Universal Robots URScript: samho_main_Fillet_2023_10_18.script

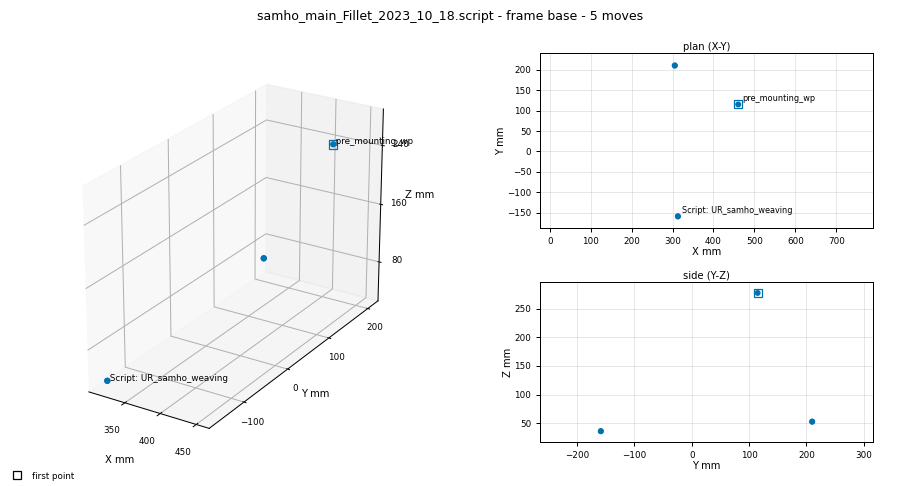
[picture p0: tool path of samho_main_Fillet_2023_10_18.script in frame base, 5 of 118 moves have a stored position in this frame; points joined in program order, loops and branches not executed]
def samho_main_Fillet_2023_10_18():
  set_standard_analog_input_domain(0, 1)
  set_standard_analog_input_domain(1, 1)
  set_tool_analog_input_domain(0, 1)
  set_tool_analog_input_domain(1, 1)
  set_analog_outputdomain(0, 1)
  set_analog_outputdomain(1, 1)
  set_input_actions_to_default()
  set_tool_digital_input_action(1, "freedrive")
  set_runstate_standard_digital_outputs([0])
  set_runstate_standard_digital_output_to_value(0, 1)
  set_runstate_standard_digital_output_to_value(7, 3)
  step_count_71f140af_8f37_405c_9852_4a67516a149e = 0.0
  thread Step_Counter_Thread_85a6b8af_9cee_45e5_b399_1c83c9369c53():
    while (True):
      step_count_71f140af_8f37_405c_9852_4a67516a149e = step_count_71f140af_8f37_405c_9852_4a67516a149e + 1.0
      sync()
    end
  end
  run Step_Counter_Thread_85a6b8af_9cee_45e5_b399_1c83c9369c53()
  modbus_add_signal("127.0.0.1", 255, 142, 2, "MODBUS_1", False)
  modbus_set_signal_update_frequency("MODBUS_1", 1)
  modbus_add_signal("127.0.0.1", 255, 152, 2, "MODBUS_2", False)
  modbus_set_signal_update_frequency("MODBUS_2", 10)
  modbus_add_signal("127.0.0.1", 255, 153, 2, "MODBUS_3", False)
  modbus_set_signal_update_frequency("MODBUS_3", 10)
  modbus_add_signal("127.0.0.1", 255, 240, 2, "MODBUS_4", False)
  modbus_set_signal_update_frequency("MODBUS_4", 10)
  set_safety_mode_transition_hardness(1)
  set_tool_voltage(24)
  set_tcp(p[-0.20862,-0.00524,0.38449,1.2551,0.019,-2.8747])
  set_payload(2.4, [-0.085, 0.00191, 0.125])
  set_gravity([0.0, 0.0, 9.82])
  global A_Touch_trig_l=[False, True, False, True, False, True, False, True, False, False, False]
  global Auto_cur_cell=0
  global last_wv_line=p[0, 0, 0, 0, 0, 0]
  global Auto_trig=True
  global A_Touch_p=[p[0, 0, 0, 0, 0, 0], p[0.49652, 0.34473, -0.02809, -1.74217, -0.74593, -1.74161], p[0, 0, 0, 0, 0, 0], p[0.50294, -0.36001, 0.02477, 1.70888, -0.78236, 1.70938], p[0, 0, 0, 0, 0, 0], p[0.49786, 0.33965, -0.0331, -1.74681, 1.75003, -0.74209], p[0, 0, 0, 0, 0, 0], p[0.50148, -0.2752, -0.03447, -1.75566, 1.75559, -0.7328], p[0, 0, 0, 0, 0, 0], p[0, 0, 0, 0, 0, 0], p[0, 0, 0, 0, 0, 0], p[0, 0, 0, 0, 0, 0], p[0, 0, 0, 0, 0, 0], p[0, 0, 0, 0, 0, 0], p[0, 0, 0, 0, 0, 0], p[0, 0, 0, 0, 0, 0]]
  global last_wv_wp1=p[0, 0, 0, 0, 0, 0]
  global last_pose=p[0, 0, 0, 0, 0, 0]
  global A_Distance_list=[0, 0, 0, 0, 0, 0, 0, 0, 0, 0, 0, 0, 0, 0, 0, 0]
  global Auto_total_cell=4
  global Reset_Trig=False
  global A_Prepos_l=[p[0, 0, 0, 0, 0, 0], p[0.46861, 0.32973, 0.0248, -2.17926, -0.88648, -1.41868], p[0, 0, 0, 0, 0, 0], p[0.46861, -0.33027, 0.0498, 1.84179, -1.10813, 1.58337], p[0, 0, 0, 0, 0, 0], p[0.47174, 0.31972, 0.02458, -2.36882, -1.02821, -1.3113], p[0, 0, 0, 0, 0, 0], p[0.46616, -0.25026, 0.02497, 2.26908, -1.08882, 1.27698], p[0, 0, 0, 0, 0, 0], p[0, 0, 0, 0, 0, 0], p[0, 0, 0, 0, 0, 0], p[0, 0, 0, 0, 0, 0], p[0, 0, 0, 0, 0, 0], p[0, 0, 0, 0, 0, 0], p[0, 0, 0, 0, 0, 0], p[0, 0, 0, 0, 0, 0]]
  global A_Speed_list=[0, 0, 0, 0, 0, 0, 0, 0, 0, 0, 0, 0, 0, 0, 0, 0]
  global Auto_W_num=[31, 32, 1, 3, 0, 0, 0, 0, 0, 0, 0, 0, 0, 0, 0]
  global last_z_bottom=-0.0502
  global last_tilt_deg=[0, 0, 0]
  global Base=p[0.0,0.0,0.0,0.0,0.0,0.0]
  global save_timer=0
  global timer_1=0
  def calculate_point_to_move_towards(feature, direction, position_distance):
    local posDir=[direction[0], direction[1], direction[2]]
    if (norm(posDir) < 1e-6):
      return get_target_waypoint()
    end
    local direction_vector_normalized=normalize(posDir)
    local displacement_pose=p[direction_vector_normalized[0] * position_distance,direction_vector_normalized[1] * position_distance,direction_vector_normalized[2] * position_distance,0,0,0]
    local wanted_displacement_in_base_frame=pose_sub(pose_trans(feature, displacement_pose), feature)
    return pose_add(get_target_waypoint(), wanted_displacement_in_base_frame)
  end
  global save_timer_is_counting=False
  global timer_1_is_counting=False
  thread Timer_Thread():
    while (True):
      if (save_timer_is_counting):
        save_timer = save_timer + get_steptime()
      end
      if (timer_1_is_counting):
        timer_1 = timer_1 + get_steptime()
      end
      sync()
    end
  end
  run Timer_Thread()
  def cell_info():
    $ 1461 "cell_info" "noBreak"
    $ 1462 "'cell_setting'"
    # 'cell_setting'
    $ 1463 "a7_f_distance≔get_center"
    global a7_f_distance=get_center
    $ 1464 "'dis + 125'"
    # 'dis + 125'
    $ 1465 "If simulation_mode"
    if (simulation_mode):
      $ 1466 "a6_f_height_l≔190"
      global a6_f_height_l=190
      $ 1467 "a6_f_height_r≔190"
      global a6_f_height_r=190
      $ 1468 "a6_f_width≔690"
      global a6_f_width=690
      $ 1469 "a6_callar_hor≔100"
      global a6_callar_hor=100
      $ 1470 "a6_callar_vert≔100"
      global a6_callar_vert=100
      $ 1471 "center_height≔50"
      global center_height=50
      $ 1472 "EXT_flag1≔integer_to_binary_list(2048)"
      global EXT_flag1= integer_to_binary_list (2048)
      $ 1473 "get_margin_z≔50"
      global get_margin_z=50
    else:
      $ 1474 "Else" "noBreak"
      $ 1475 "a6_f_height_l≔read_port_register(173)"
      global a6_f_height_l= read_port_register (173)
      $ 1476 "a6_f_height_r≔read_port_register(174)"
      global a6_f_height_r= read_port_register (174)
      $ 1477 "a6_f_width≔read_port_register(175)"
      global a6_f_width= read_port_register (175)
      $ 1478 "a6_callar_hor≔read_port_register(181)"
      global a6_callar_hor= read_port_register (181)
      $ 1479 "a6_callar_vert≔read_port_register(182)"
      global a6_callar_vert= read_port_register (182)
      $ 1480 "center_height≔read_port_register(237)"
      global center_height=read_port_register(237)
      $ 1481 "EXT_flag1≔integer_to_binary_list(read_port_register(179))"
      global EXT_flag1= integer_to_binary_list ( read_port_register (179))
      $ 1483 "get_margin_z≔read_port_register(238)"
      global get_margin_z=read_port_register(238)
      $ 1485 "If center_height>32765"
      if (center_height>32765):
        $ 1486 "center_height≔center_height-65535"
        global center_height=center_height-65535
      end
      $ 1487 "If get_margin_z>32765"
      if (get_margin_z>32765):
        $ 1488 "get_margin_z≔get_margin_z-65535"
        global get_margin_z=get_margin_z-65535
      end
    end
    $ 1489 "Initialization"
    $ 1490 "CELL_ROBOT_DIST≔a7_f_distance"
    global CELL_ROBOT_DIST=a7_f_distance
    $ 1491 "CELL_WIDTH≔a6_f_width"
    global CELL_WIDTH=a6_f_width
  end
  def robotand_cell_initalizat():
    $ 1492 "robotand_cell_initalizat" "noBreak"
    $ 1493 "If Auto_trig≟ True "
    if (Auto_trig ==   True  ):
      $ 1494 "Auto_trig≔ False "
      global Auto_trig=  False
      $ 1495 "init"
      $ 1496 "write_port_register(cell_3f_2f_151,0)"
      write_port_register(cell_3f_2f_151,0)
      $ 1497 "write_port_register(cell_info_152,0)"
      write_port_register(cell_info_152,0)
      $ 1498 "write_port_register(weld_req_153,0)"
      write_port_register(weld_req_153,0)
      $ 1499 "write_port_register(touch_cell_155,0)"
      write_port_register(touch_cell_155,0)
      $ 1500 "write_port_register(touch_num_156,0)"
      write_port_register(touch_num_156,0)
      $ 1501 "write_port_register(touch_done_157,0)"
      write_port_register(touch_done_157,0)
      $ 1502 "write_port_register(weld_done_137,0)"
      write_port_register(weld_done_137,0)
      $ 1503 "write_port_register(135,0)"
      write_port_register(135,0)
      $ 1504 "write_port_register(136,0)"
      write_port_register(136,0)
      $ 1505 "write_port_register(165,0)"
      write_port_register(165,0)
      $ 1506 "write_port_register(166,0)"
      write_port_register(166,0)
      $ 1507 "write_port_register(167,0)"
      write_port_register(167,0)
      $ 1508 "write_port_register(169,0)"
      write_port_register(169,0)
      $ 1509 "write_port_register(170,0)"
      write_port_register(170,0)
      $ 1510 "write_port_register(221,0)"
      write_port_register(221,0)
      $ 1511 "write_port_register(222,0)"
      write_port_register(222,0)
      $ 1512 "write_port_register(223,0)"
      write_port_register(223,0)
      $ 1513 "write_port_register(224,0)"
      write_port_register(224,0)
      $ 1514 "write_port_register(225,0)"
      write_port_register(225,0)
      $ 1515 "write_port_register(226,0)"
      write_port_register(226,0)
      $ 1516 "write_port_register(227,0)"
      write_port_register(227,0)
      $ 1517 "write_port_register(228,0)"
      write_port_register(228,0)
      $ 1518 "write_port_register(240,0)"
      write_port_register(240,0)
      $ 1519 "write_port_register(176,0)"
      write_port_register(176,0)
      $ 1520 "write_port_register(177,0)"
      write_port_register(177,0)
      $ 1521 "write_port_register(154,0)"
      write_port_register(154,0)
    end
    $ 1522 "sync()"
    sync()
  end
  def welding_parameter_init():
    $ 1523 "welding_parameter_init" "noBreak"
    $ 1524 "init"
    $ 1525 "If A_sel_v≟A_VL1 or A_sel_v≟A_VL2 or A_sel_v≟A_VR1 or A_sel_v≟A_VR2"
    if (A_sel_v == A_VL1  or  A_sel_v == A_VL2  or  A_sel_v == A_VR1  or  A_sel_v == A_VR2):
      $ 1526 "position_3f2f≔position_3F"
      global position_3f2f=position_3F
      $ 1527 "write_port_register(cell_3f_2f_151,A_sel_v)"
      write_port_register(cell_3f_2f_151,A_sel_v)
      $ 1528 "b8_wv_2f≔ False "
      global b8_wv_2f=  False
      $ 1529 "d_lean_degree≔0"
      global d_lean_degree=0
    else:
      $ 1530 "Else" "noBreak"
      $ 1531 "position_3f2f≔position_2F"
      global position_3f2f=position_2F
      $ 1532 "b8_wv_2f≔ True "
      global b8_wv_2f=  True
      $ 1533 "d_lean_degree≔30"
      global d_lean_degree=30
      $ 1534 "write_port_register(cell_3f_2f_151,A_HOR)"
      write_port_register(cell_3f_2f_151,A_HOR)
    end
    $ 1535 "If current_path≥2"
    if (current_path >= 2):
      $ 1536 "write_port_register(cell_info_152,current_path)"
      write_port_register(cell_info_152,current_path)
    else:
      $ 1537 "Else" "noBreak"
      $ 1538 "write_port_register(cell_info_152,1)"
      write_port_register(cell_info_152,1)
    end
    $ 1539 "write_port_register(return_done_240,0)"
    write_port_register(return_done_240,0)
    $ 1540 "Wait: 0.3"
    sleep(0.3)
    $ 1541 "write_port_register(weld_req_153,1)"
    write_port_register(weld_req_153,1)
    $ 1542 "Wait read_port_register(return_done_240)≟1"
    while (not( read_port_register (return_done_240) == 1)):
      sync()
    end
    $ 1543 "write_port_register(weld_req_153,0)"
    write_port_register(weld_req_153,0)
    $ 1544 "touch_m_check≔0"
    global touch_m_check=0
    $ 1545 "start_end_from_pendant"
    $ 1546 "d_start_current≔read_port_register(244)/10"
    global d_start_current= read_port_register (244)/10
    $ 1547 "d_start_voltage≔read_port_register(245)/10"
    global d_start_voltage= read_port_register (245)/10
    $ 1548 "d_start_time≔read_port_register(241)/10"
    global d_start_time= read_port_register (241)/10
    $ 1549 "d_end_current≔read_port_register(249)/10"
    global d_end_current= read_port_register (249)/10
    $ 1550 "d_end_voltage≔read_port_register(250)/10"
    global d_end_voltage= read_port_register (250)/10
    $ 1551 "d_end_time≔read_port_register(246)/10"
    global d_end_time= read_port_register (246)/10
    $ 1552 "d_end_current_2≔read_port_register(254)/10"
    global d_end_current_2= read_port_register (254)/10
    $ 1553 "d_end_voltage_2≔read_port_register(255)/10"
    global d_end_voltage_2= read_port_register (255)/10
    $ 1554 "d_end_time_2≔read_port_register(251)/10"
    global d_end_time_2= read_port_register (251)/10
    $ 1555 "a7_weld_crater≔[d_start_current,d_start_voltage,d_start_time,d_end_current,d_end_voltage,d_end_time,d_lean_degree]"
    global a7_weld_crater=[d_start_current,d_start_voltage,d_start_time,d_end_current,d_end_voltage,d_end_time,d_lean_degree]
    $ 1556 "a0_volt_ref≔read_port_register(231)/10"
    global a0_volt_ref= read_port_register (231)/10
    $ 1557 "a1_amp_ref≔read_port_register(232)/10"
    global a1_amp_ref= read_port_register (232)/10
    $ 1558 "a2_speed_cpm≔read_port_register(233)/10"
    global a2_speed_cpm= read_port_register (233)/10
    $ 1559 "a3_wv_amplitude≔read_port_register(234)/10"
    global a3_wv_amplitude= read_port_register (234)/10
    $ 1560 "a4_wv_frequency≔read_port_register(225)/10"
    global a4_wv_frequency= read_port_register (225)/10
    $ 1561 "b1_appro_param≔0"
    global b1_appro_param=0
    $ 1562 "b4_wv_delay2≔read_port_register(226)/10"
    global b4_wv_delay2= read_port_register (226)/10
    $ 1563 "b6_wv_delay4≔read_port_register(227)/10"
    global b6_wv_delay4= read_port_register (227)/10
    $ 1564 "b3_wv_delay1≔0"
    global b3_wv_delay1=0
    $ 1565 "b5_wv_delay3≔0"
    global b5_wv_delay3=0
    $ 1566 "b3_dealy_all≔[b3_wv_delay1,b4_wv_delay2,b5_wv_delay3,b6_wv_delay4]"
    global b3_dealy_all=[b3_wv_delay1,b4_wv_delay2,b5_wv_delay3,b6_wv_delay4]
    $ 1567 "get_width_182≔read_port_register(182)"
    global get_width_182= read_port_register (182)
    $ 1568 "b9_touch_sens≔20"
    global b9_touch_sens=20
    $ 1569 "task_angle≔register_read(228)/10"
    global task_angle=register_read(228)/10
    $ 1570 "Circle_Speed≔a2_speed_cpm"
    global Circle_Speed=a2_speed_cpm
    $ 1571 "CELL_BOTTOM≔a7_cell_bottom"
    global CELL_BOTTOM=a7_cell_bottom
    $ 1572 "a6_scallup_left≔read_port_register(176)"
    global a6_scallup_left= read_port_register (176)
    $ 1573 "a6_scallup_righ≔read_port_register(177)"
    global a6_scallup_righ= read_port_register (177)
    $ 1574 "a5_f_hole≔[a7_cell_bottom,a6_scallup_left,a6_scallup_righ]"
    global a5_f_hole=[a7_cell_bottom,a6_scallup_left,a6_scallup_righ]
    $ 1608 "폴더"
    $ 1609 "offset_2f_x≔7"
    global offset_2f_x=7
    $ 1610 "offset_3f_z≔-5"
    global offset_3f_z=-5
    $ 1611 "If A_sel_v≟A_VR1 or A_sel_v≟A_VR2"
    if (A_sel_v == A_VR1  or  A_sel_v == A_VR2):
      $ 1612 "'3F'"
      # '3F'
      $ 1613 "b2_left_par≔ False "
      global b2_left_par=  False
      $ 1614 "b8_wv_type≔1"
      global b8_wv_type=1
      $ 1615 "If A_sel_v≟A_VR2 and (b1_cell_info_R≟c or b1_cell_info_R≟d)"
      if (A_sel_v == A_VR2  and  (b1_cell_info_R == c  or  b1_cell_info_R == d)):
        $ 1616 "b7_tilt_degree≔[0,0,0]"
        global b7_tilt_degree=[0,0,0]
      else:
        $ 1617 "Else" "noBreak"
        $ 1618 "b7_tilt_degree≔[task_angle,-27,0]"
        global b7_tilt_degree=[task_angle,-27,0]
      end
      $ 1619 "c3_arc_enable≔1"
      global c3_arc_enable=1
    else:
      $ 1620 "ElseIf A_sel_v≟A_VL1 or A_sel_v≟A_VL2"
      if (A_sel_v == A_VL1  or  A_sel_v == A_VL2):
        $ 1621 "'3F'"
        # '3F'
        $ 1622 "b2_left_par≔ True "
        global b2_left_par=  True
        $ 1623 "b8_wv_type≔1"
        global b8_wv_type=1
        $ 1624 "If A_sel_v≟A_VL2 and (b1_cell_info_L≟c or b1_cell_info_L≟d)"
        if (A_sel_v == A_VL2  and  (b1_cell_info_L == c  or  b1_cell_info_L == d)):
          $ 1625 "b7_tilt_degree≔[0,0,0]"
          global b7_tilt_degree=[0,0,0]
        else:
          $ 1626 "Else" "noBreak"
          $ 1627 "b7_tilt_degree≔[task_angle,-27,0]"
          global b7_tilt_degree=[task_angle,-27,0]
        end
        $ 1628 "c3_arc_enable≔1"
        global c3_arc_enable=1
      else:
        $ 1629 "Else" "noBreak"
        $ 1630 "b2_left_par≔ True "
        global b2_left_par=  True
        $ 1631 "b8_wv_type≔2"
        global b8_wv_type=2
        $ 1632 "If A_sel_v≟A_HOR"
        if (A_sel_v == A_HOR):
          $ 1633 "b7_tilt_degree≔[30,-1*task_angle,0]"
          global b7_tilt_degree=[30,-1*task_angle,0]
        else:
          $ 1634 "Else" "noBreak"
          $ 1636 "b7_tilt_degree≔[30,-1*task_angle,0]"
          global b7_tilt_degree=[30,-1*task_angle,0]
        end
        $ 1638 "c3_arc_enable≔0"
        global c3_arc_enable=0
      end
    end
    $ 1639 "If A_sel_v≟A_VL2 or A_sel_v≟A_VR2"
    if (A_sel_v == A_VL2  or  A_sel_v == A_VR2):
      $ 1640 "a8_wv_distance≔read_port_register(182)-offset_3f_begin"
      global a8_wv_distance= read_port_register (182)-offset_3f_begin
    else:
      $ 1645 "Else" "noBreak"
      $ 1646 "If b2_left_par"
      if (b2_left_par):
        $ 1647 "Comment"
        # Comment
        $ 1648 "a8_wv_distance≔a6_f_height_l-a5_f_hole[1]-offset_3f_begin"
        global a8_wv_distance=a6_f_height_l-a5_f_hole[1]-offset_3f_begin
        $ 1649 "Comment"
        # Comment
      else:
        $ 1650 "Else" "noBreak"
        $ 1651 "a8_wv_distance≔a6_f_height_r-a5_f_hole[1]-offset_3f_begin"
        global a8_wv_distance=a6_f_height_r-a5_f_hole[1]-offset_3f_begin
      end
    end
    $ 1652 "Ext fun & Squash"
    $ 1653 "If (A_sel_v≟A_VL1 or A_sel_v≟A_VL2) and (b1_cell_info_L≟B or b1_cell_info_L≟D)"
    if ((A_sel_v == A_VL1  or  A_sel_v == A_VL2)  and  (b1_cell_info_L == B  or  b1_cell_info_L == D)):
      $ 1654 "Scallup_check≔ True "
      global Scallup_check=  True
    else:
      $ 1655 "ElseIf (A_sel_v≟A_VR1 or A_sel_v≟A_VR2) and (b1_cell_info_R≟B or b1_cell_info_R≟D)"
      if ((A_sel_v == A_VR1  or  A_sel_v == A_VR2)  and  (b1_cell_info_R == B  or  b1_cell_info_R == D)):
        $ 1656 "Scallup_check≔ True "
        global Scallup_check=  True
      else:
        $ 1657 "Else" "noBreak"
        $ 1658 "Scallup_check≔ False "
        global Scallup_check=  False
      end
    end
    $ 1659 "If (EXT_flag1[7]≟ True ) and (A_sel_v≠A_HOR) and (A_sel_v≠A_VL2) and (A_sel_v≠A_VR2) and (Scallup_check≟ False )"
    if ((EXT_flag1[7] ==   True  )  and  (A_sel_v != A_HOR)  and  (A_sel_v != A_VL2)  and  (A_sel_v != A_VR2)  and  (Scallup_check ==   False  )):
      $ 1660 "squash"
      $ 1661 "squash_enable≔1"
      global squash_enable=1
      $ 1662 "squash_voltage≔24.5"
      global squash_voltage=24.5
      $ 1663 "squash_current≔190"
      global squash_current=190
      $ 1664 "squash_amp≔7"
      global squash_amp=7
      $ 1665 "squash_speed≔10"
      global squash_speed=10
      $ 1666 "squash_cycle≔8"
      global squash_cycle=8
    else:
      $ 1667 "Else" "noBreak"
      $ 1668 "squash"
      $ 1669 "squash_enable≔0"
      global squash_enable=0
      $ 1670 "squash_voltage≔0"
      global squash_voltage=0
      $ 1671 "squash_current≔0"
      global squash_current=0
      $ 1672 "squash_amp≔0"
      global squash_amp=0
      $ 1673 "squash_speed≔0"
      global squash_speed=0
      $ 1674 "squash_cycle≔0"
      global squash_cycle=0
    end
    $ 1675 "If EXT_flag1[8]≟ True  and EXT_flag1[9]≟ False "
    if (EXT_flag1[8] ==   True    and  EXT_flag1[9] ==   False  ):
      $ 1676 "sludge≔1"
      global sludge=1
    else:
      $ 1677 "ElseIf EXT_flag1[8]≟ False  and EXT_flag1[9]≟ True "
      if (EXT_flag1[8] ==   False    and  EXT_flag1[9] ==   True  ):
        $ 1678 "sludge≔2"
        global sludge=2
      else:
        $ 1679 "Else" "noBreak"
        $ 1680 "sludge≔0"
        global sludge=0
      end
    end
    $ 1681 "waste_cycle≔2"
    global waste_cycle=2
    $ 1682 "c0_offset_x≔read_port_register(229)/10"
    global c0_offset_x= read_port_register (229)/10
    $ 1683 "c0_offset_z≔read_port_register(230)/10"
    global c0_offset_z= read_port_register (230)/10
    $ 1684 "squash_l≔[a0_volt_ref,a1_amp_ref,squash_enable,squash_voltage,squash_current,squash_amp,squash_speed,squash_cycle,waste_cycle,c0_offset_x,c0_offset_z]"
    global squash_l=[a0_volt_ref,a1_amp_ref,squash_enable,squash_voltage,squash_current,squash_amp,squash_speed,squash_cycle,waste_cycle,c0_offset_x,c0_offset_z]
    $ 1685 "WV_gap"
    $ 1686 "c5_wv_gap_y≔read_port_register(236)/10"
    global c5_wv_gap_y= read_port_register (236)/10
    $ 1687 "c6_wv_gap_cpm≔read_port_register(235)/10"
    global c6_wv_gap_cpm= read_port_register (235)/10
    $ 1688 "c9_wv_gap_freq≔a4_wv_frequency"
    global c9_wv_gap_freq=a4_wv_frequency
    $ 1689 "If c6_wv_gap_cpm≟a2_speed_cpm and a3_wv_amplitude≟c5_wv_gap_y"
    if (c6_wv_gap_cpm == a2_speed_cpm  and  a3_wv_amplitude == c5_wv_gap_y):
      $ 1690 "c4_gap_enable≔0"
      global c4_gap_enable=0
    else:
      $ 1691 "Else" "noBreak"
      $ 1692 "c4_gap_enable≔1"
      global c4_gap_enable=1
    end
    $ 1693 "c7_wv_gap≔[c4_gap_enable,c5_wv_gap_y,c6_wv_gap_cpm,c9_wv_gap_freq]"
    global c7_wv_gap=[c4_gap_enable,c5_wv_gap_y,c6_wv_gap_cpm,c9_wv_gap_freq]
    $ 1694 "arc_sen"
    $ 1695 "c3_X_p_gain≔read_port_register(186)/10"
    global c3_X_p_gain= read_port_register (186)/10
    $ 1696 "c3_X_i_gain≔read_port_register(187)/10"
    global c3_X_i_gain= read_port_register (187)/10
    $ 1697 "c3_Z_p_gain≔read_port_register(184)/10"
    global c3_Z_p_gain= read_port_register (184)/10
    $ 1698 "c3_Z_i_gain≔read_port_register(185)/10"
    global c3_Z_i_gain= read_port_register (185)/10
    $ 1699 "c3_wv_arc_fix≔0"
    global c3_wv_arc_fix=0
    $ 1700 "c3_wv_arc≔[c3_arc_enable,c3_X_p_gain,c3_X_i_gain,c3_Z_p_gain,c3_Z_i_gain,c3_wv_arc_fix]"
    global c3_wv_arc=[c3_arc_enable,c3_X_p_gain,c3_X_i_gain,c3_Z_p_gain,c3_Z_i_gain,c3_wv_arc_fix]
    $ 1701 "volt and current"
    $ 1702 "set_current_voltage(a1_amp_ref,a0_volt_ref)"
    set_current_voltage(a1_amp_ref,a0_volt_ref)
    $ 1703 "write_port_register(154,1)"
    write_port_register(154,1)
    $ 1704 "Wait read_port_register(return_done_240)≟0"
    while (not( read_port_register (return_done_240) == 0)):
      sync()
    end
    $ 1705 "write_port_register(154,0)"
    write_port_register(154,0)
  end
  def welding_parameter_sim():
    $ 1706 "welding_parameter_sim" "noBreak"
    $ 1707 "init"
    $ 1708 "If A_sel_v≟A_VL1 or A_sel_v≟A_VL2 or A_sel_v≟A_VR1 or A_sel_v≟A_VR2"
    if (A_sel_v == A_VL1  or  A_sel_v == A_VL2  or  A_sel_v == A_VR1  or  A_sel_v == A_VR2):
      $ 1709 "position_3f2f≔position_3F"
      global position_3f2f=position_3F
      $ 1710 "write_port_register(cell_3f_2f_151,A_sel_v)"
      write_port_register(cell_3f_2f_151,A_sel_v)
      $ 1711 "b8_wv_2f≔ False "
      global b8_wv_2f=  False
      $ 1712 "d_lean_degree≔0"
      global d_lean_degree=0
    else:
      $ 1713 "Else" "noBreak"
      $ 1714 "position_3f2f≔position_2F"
      global position_3f2f=position_2F
      $ 1715 "b8_wv_2f≔ True "
      global b8_wv_2f=  True
      $ 1716 "d_lean_degree≔30"
      global d_lean_degree=30
      $ 1717 "write_port_register(cell_3f_2f_151,A_HOR)"
      write_port_register(cell_3f_2f_151,A_HOR)
    end
    $ 1718 "If current_path≥2"
    if (current_path >= 2):
      $ 1719 "write_port_register(cell_info_152,current_path)"
      write_port_register(cell_info_152,current_path)
    else:
      $ 1720 "Else" "noBreak"
      $ 1721 "write_port_register(cell_info_152,1)"
      write_port_register(cell_info_152,1)
    end
    $ 1722 "write_port_register(return_done_240,0)"
    write_port_register(return_done_240,0)
    $ 1723 "Wait: 0.3"
    sleep(0.3)
    $ 1724 "write_port_register(weld_req_153,1)"
    write_port_register(weld_req_153,1)
    $ 1726 "write_port_register(weld_req_153,0)"
    write_port_register(weld_req_153,0)
    $ 1727 "touch_m_check≔0"
    global touch_m_check=0
    $ 1728 "start_end_from_pendant"
    $ 1729 "d_start_current≔read_port_register(244)/10"
    global d_start_current= read_port_register (244)/10
    $ 1730 "d_start_voltage≔read_port_register(245)/10"
    global d_start_voltage= read_port_register (245)/10
    $ 1731 "d_start_time≔read_port_register(241)/10"
    global d_start_time= read_port_register (241)/10
    $ 1732 "d_end_current≔read_port_register(249)/10"
    global d_end_current= read_port_register (249)/10
    $ 1733 "d_end_voltage≔read_port_register(250)/10"
    global d_end_voltage= read_port_register (250)/10
    $ 1734 "d_end_time≔read_port_register(246)/10"
    global d_end_time= read_port_register (246)/10
    $ 1735 "d_end_current_2≔read_port_register(254)/10"
    global d_end_current_2= read_port_register (254)/10
    $ 1736 "d_end_voltage_2≔read_port_register(255)/10"
    global d_end_voltage_2= read_port_register (255)/10
    $ 1737 "d_end_time_2≔read_port_register(251)/10"
    global d_end_time_2= read_port_register (251)/10
    $ 1738 "a7_weld_crater≔[d_start_current,d_start_voltage,d_start_time,d_end_current,d_end_voltage,d_end_time,d_lean_degree]"
    global a7_weld_crater=[d_start_current,d_start_voltage,d_start_time,d_end_current,d_end_voltage,d_end_time,d_lean_degree]
    $ 1739 "a0_volt_ref≔read_port_register(231)/10"
    global a0_volt_ref= read_port_register (231)/10
    $ 1740 "a1_amp_ref≔read_port_register(232)/10"
    global a1_amp_ref= read_port_register (232)/10
    $ 1741 "b1_appro_param≔0"
    global b1_appro_param=0
    $ 1742 "Folder"
    $ 1743 "a2_speed_cpm≔17"
    global a2_speed_cpm=17
    $ 1744 "a3_wv_amplitude≔5"
    global a3_wv_amplitude=5
    $ 1745 "a4_wv_frequency≔1.4"
    global a4_wv_frequency=1.4
    $ 1746 "b4_wv_delay2≔0.3"
    global b4_wv_delay2=0.3
    $ 1747 "b6_wv_delay4≔0.3"
    global b6_wv_delay4=0.3
    $ 1748 "b9_touch_sens≔10"
    global b9_touch_sens=10
    $ 1749 "task_angle≔0"
    global task_angle=0
    $ 1750 "a6_scallup_left≔0"
    global a6_scallup_left=0
    $ 1751 "a6_scallup_righ≔0"
    global a6_scallup_righ=0
    $ 1752 "b3_wv_delay1≔0"
    global b3_wv_delay1=0
    $ 1753 "b5_wv_delay3≔0"
    global b5_wv_delay3=0
    $ 1754 "b3_dealy_all≔[b3_wv_delay1,b4_wv_delay2,b5_wv_delay3,b6_wv_delay4]"
    global b3_dealy_all=[b3_wv_delay1,b4_wv_delay2,b5_wv_delay3,b6_wv_delay4]
    $ 1755 "get_width_182≔a6_callar_vert"
    global get_width_182=a6_callar_vert
    $ 1756 "task_angle≔register_read(228)/10"
    global task_angle=register_read(228)/10
    $ 1757 "Circle_Speed≔a2_speed_cpm"
    global Circle_Speed=a2_speed_cpm
    $ 1758 "CELL_BOTTOM≔a7_cell_bottom"
    global CELL_BOTTOM=a7_cell_bottom
    $ 1759 "a5_f_hole≔[a7_cell_bottom,a6_scallup_left,a6_scallup_righ]"
    global a5_f_hole=[a7_cell_bottom,a6_scallup_left,a6_scallup_righ]
    $ 1760 "폴더"
    $ 1761 "offset_2f_x≔7"
    global offset_2f_x=7
    $ 1762 "offset_3f_z≔-5"
    global offset_3f_z=-5
    $ 1763 "If A_sel_v≟A_VR1 or A_sel_v≟A_VR2"
    if (A_sel_v == A_VR1  or  A_sel_v == A_VR2):
      $ 1764 "'3F'"
      # '3F'
      $ 1765 "b2_left_par≔ False "
      global b2_left_par=  False
      $ 1766 "b8_wv_type≔1"
      global b8_wv_type=1
      $ 1767 "b7_tilt_degree≔[task_angle,-27,0]"
      global b7_tilt_degree=[task_angle,-27,0]
      $ 1768 "c3_arc_enable≔1"
      global c3_arc_enable=1
    else:
      $ 1769 "ElseIf A_sel_v≟A_VL1 or A_sel_v≟A_VL2"
      if (A_sel_v == A_VL1  or  A_sel_v == A_VL2):
        $ 1770 "'3F'"
        # '3F'
        $ 1771 "b2_left_par≔ True "
        global b2_left_par=  True
        $ 1772 "b8_wv_type≔1"
        global b8_wv_type=1
        $ 1773 "b7_tilt_degree≔[task_angle,-27,0]"
        global b7_tilt_degree=[task_angle,-27,0]
        $ 1774 "c3_arc_enable≔1"
        global c3_arc_enable=1
      else:
        $ 1775 "Else" "noBreak"
        $ 1776 "b2_left_par≔ True "
        global b2_left_par=  True
        $ 1777 "b8_wv_type≔2"
        global b8_wv_type=2
        $ 1778 "b7_tilt_degree≔[30,-1*task_angle,0]"
        global b7_tilt_degree=[30,-1*task_angle,0]
        $ 1780 "c3_arc_enable≔0"
        global c3_arc_enable=0
      end
    end
    $ 1781 "If A_sel_v≟A_VL2 or A_sel_v≟A_VR2"
    if (A_sel_v == A_VL2  or  A_sel_v == A_VR2):
      $ 1782 "a8_wv_distance≔read_port_register(182)"
      global a8_wv_distance= read_port_register (182)
    else:
      $ 1787 "Else" "noBreak"
      $ 1788 "If b2_left_par"
      if (b2_left_par):
        $ 1789 "Comment"
        # Comment
        $ 1790 "a8_wv_distance≔a6_f_height_l-a5_f_hole[1]"
        global a8_wv_distance=a6_f_height_l-a5_f_hole[1]
        $ 1791 "Comment"
        # Comment
      else:
        $ 1792 "Else" "noBreak"
        $ 1793 "a8_wv_distance≔a6_f_height_r-a5_f_hole[1]"
        global a8_wv_distance=a6_f_height_r-a5_f_hole[1]
      end
    end
    $ 1794 "Ext fun & Squash"
    $ 1795 "If (A_sel_v≟A_VL1 or A_sel_v≟A_VL2) and (b1_cell_info_L≟B or b1_cell_info_L≟D)"
    if ((A_sel_v == A_VL1  or  A_sel_v == A_VL2)  and  (b1_cell_info_L == B  or  b1_cell_info_L == D)):
      $ 1796 "Scallup_check≔ True "
      global Scallup_check=  True
    else:
      $ 1797 "ElseIf (A_sel_v≟A_VR1 or A_sel_v≟A_VR2) and (b1_cell_info_R≟B or b1_cell_info_R≟D)"
      if ((A_sel_v == A_VR1  or  A_sel_v == A_VR2)  and  (b1_cell_info_R == B  or  b1_cell_info_R == D)):
        $ 1798 "Scallup_check≔ True "
        global Scallup_check=  True
      else:
        $ 1799 "Else" "noBreak"
        $ 1800 "Scallup_check≔ False "
        global Scallup_check=  False
      end
    end
    $ 1801 "If (EXT_flag1[7]≟ True ) and (A_sel_v≠A_HOR) and (A_sel_v≠A_VL2) and (A_sel_v≠A_VR2) and (Scallup_check≟ False )"
    if ((EXT_flag1[7] ==   True  )  and  (A_sel_v != A_HOR)  and  (A_sel_v != A_VL2)  and  (A_sel_v != A_VR2)  and  (Scallup_check ==   False  )):
      $ 1802 "squash"
      $ 1803 "squash_enable≔1"
      global squash_enable=1
      $ 1804 "squash_voltage≔24.5"
      global squash_voltage=24.5
      $ 1805 "squash_current≔190"
      global squash_current=190
      $ 1806 "squash_amp≔7"
      global squash_amp=7
      $ 1807 "squash_speed≔10"
      global squash_speed=10
      $ 1808 "squash_cycle≔8"
      global squash_cycle=8
    else:
      $ 1809 "Else" "noBreak"
      $ 1810 "squash"
      $ 1811 "squash_enable≔0"
      global squash_enable=0
      $ 1812 "squash_voltage≔0"
      global squash_voltage=0
      $ 1813 "squash_current≔0"
      global squash_current=0
      $ 1814 "squash_amp≔0"
      global squash_amp=0
      $ 1815 "squash_speed≔0"
      global squash_speed=0
      $ 1816 "squash_cycle≔0"
      global squash_cycle=0
    end
    $ 1817 "waste_cycle≔2"
    global waste_cycle=2
    $ 1818 "c0_offset_x≔read_port_register(229)/10"
    global c0_offset_x= read_port_register (229)/10
    $ 1819 "c0_offset_z≔read_port_register(230)/10"
    global c0_offset_z= read_port_register (230)/10
    $ 1820 "squash_l≔[a0_volt_ref,a1_amp_ref,squash_enable,squash_voltage,squash_current,squash_amp,squash_speed,squash_cycle,waste_cycle,c0_offset_x,c0_offset_z]"
    global squash_l=[a0_volt_ref,a1_amp_ref,squash_enable,squash_voltage,squash_current,squash_amp,squash_speed,squash_cycle,waste_cycle,c0_offset_x,c0_offset_z]
    $ 1821 "WV_gap"
    $ 1822 "c5_wv_gap_y≔a3_wv_amplitude"
    global c5_wv_gap_y=a3_wv_amplitude
    $ 1823 "c6_wv_gap_cpm≔a2_speed_cpm"
    global c6_wv_gap_cpm=a2_speed_cpm
    $ 1824 "c9_wv_gap_freq≔a4_wv_frequency"
    global c9_wv_gap_freq=a4_wv_frequency
    $ 1825 "If c6_wv_gap_cpm≟a2_speed_cpm and a3_wv_amplitude≟c5_wv_gap_y"
    if (c6_wv_gap_cpm == a2_speed_cpm  and  a3_wv_amplitude == c5_wv_gap_y):
      $ 1826 "c4_gap_enable≔0"
      global c4_gap_enable=0
    else:
      $ 1827 "Else" "noBreak"
      $ 1828 "c4_gap_enable≔1"
      global c4_gap_enable=1
    end
    $ 1829 "c4_gap_enable≔0"
    global c4_gap_enable=0
    $ 1830 "c7_wv_gap≔[c4_gap_enable,c5_wv_gap_y,c6_wv_gap_cpm,c9_wv_gap_freq]"
    global c7_wv_gap=[c4_gap_enable,c5_wv_gap_y,c6_wv_gap_cpm,c9_wv_gap_freq]
    $ 1831 "arc_sen"
    $ 1832 "c3_X_p_gain≔read_port_register(186)/10"
    global c3_X_p_gain= read_port_register (186)/10
    $ 1833 "c3_X_i_gain≔read_port_register(187)/10"
    global c3_X_i_gain= read_port_register (187)/10
    $ 1834 "c3_Z_p_gain≔read_port_register(184)/10"
    global c3_Z_p_gain= read_port_register (184)/10
    $ 1835 "c3_Z_i_gain≔read_port_register(185)/10"
    global c3_Z_i_gain= read_port_register (185)/10
    $ 1836 "c3_wv_arc_fix≔0"
    global c3_wv_arc_fix=0
    $ 1837 "c3_wv_arc≔[c3_arc_enable,c3_X_p_gain,c3_X_i_gain,c3_Z_p_gain,c3_Z_i_gain,c3_wv_arc_fix]"
    global c3_wv_arc=[c3_arc_enable,c3_X_p_gain,c3_X_i_gain,c3_Z_p_gain,c3_Z_i_gain,c3_wv_arc_fix]
    $ 1838 "volt and current"
    $ 1839 "set_current_voltage(a1_amp_ref,a0_volt_ref)"
    set_current_voltage(a1_amp_ref,a0_volt_ref)
    $ 1840 "write_port_register(154,1)"
    write_port_register(154,1)
    $ 1842 "write_port_register(154,0)"
    write_port_register(154,0)
  end
  def Move_done():
    $ 1843 "Move_done" "noBreak"
    $ 1844 "write_port_register(robot_move_163,0)"
    write_port_register(robot_move_163,0)
    $ 1845 "write_port_register(robot_pose_164,0)"
    write_port_register(robot_pose_164,0)
    $ 1846 "write_port_register(robot_ready_141,1)"
    write_port_register(robot_ready_141,1)
  end
  def MoveFun():
    $ 1847 "MoveFun" "noBreak"
    $ 1848 "b_touch_pos≔A_Prepos_l[A_sel_v]"
    global b_touch_pos=A_Prepos_l[A_sel_v]
    $ 1849 "MoveL"
    $ 1850 "b_touch_pos" "breakAfter"
    movel(pose_trans(Base, b_touch_pos), a=0.35, v=0.35)
  end
  def MoveFun_cd():
    $ 1851 "MoveFun_cd" "noBreak"
    $ 1852 "b_touch_pos≔A_Prepos_l[A_sel_v]"
    global b_touch_pos=A_Prepos_l[A_sel_v]
    $ 1853 "If A_sel_v≟A_VR2 and (b1_cell_info_R≟c or b1_cell_info_R≟d)"
    if (A_sel_v == A_VR2  and  (b1_cell_info_R == c  or  b1_cell_info_R == d)):
      $ 1854 "tilt_deg≔27"
      global tilt_deg=27
      $ 1855 "tilt_deg_ry≔19"
      global tilt_deg_ry=19
      $ 1856 "tilt_deg_rz≔0"
      global tilt_deg_rz=0
    else:
      $ 1857 "Else" "noBreak"
      $ 1858 "tilt_deg≔10"
      global tilt_deg=10
      $ 1859 "tilt_deg_ry≔5"
      global tilt_deg_ry=5
      $ 1860 "tilt_deg_rz≔0"
      global tilt_deg_rz=0
    end
    $ 1861 "If b2_left_par"
    if (b2_left_par):
      $ 1862 "b_touch_pos≔pose_add(b_touch_pos, p[0,18/1000,0,0,0,0])"
      global b_touch_pos= pose_add (b_touch_pos, p[0,18/1000,0,0,0,0])
      $ 1863 "b_touch_pos≔pose_trans(b_touch_pos, p[0,0,0,d2r(-tilt_deg),d2r(-tilt_deg_ry),d2r(tilt_deg_rz)])"
      global b_touch_pos= pose_trans (b_touch_pos, p[0,0,0,d2r(-tilt_deg),d2r(-tilt_deg_ry),d2r(tilt_deg_rz)])
    else:
      $ 1864 "Else" "noBreak"
      $ 1865 "b_touch_pos≔pose_add(b_touch_pos, p[0,-18/1000,0,0,0,0])"
      global b_touch_pos= pose_add (b_touch_pos, p[0,-18/1000,0,0,0,0])
      $ 1866 "b_touch_pos≔pose_trans(b_touch_pos, p[0,0,0,d2r(tilt_deg),d2r(-tilt_deg_ry),d2r(-tilt_deg_rz)])"
      global b_touch_pos= pose_trans (b_touch_pos, p[0,0,0,d2r(tilt_deg),d2r(-tilt_deg_ry),d2r(-tilt_deg_rz)])
    end
    $ 1867 "MoveL"
    $ 1868 "b_touch_pos" "breakAfter"
    movel(pose_trans(Base, b_touch_pos), a=0.35, v=0.35)
  end
  def MoveandTouchFun_2f():
    $ 1869 "MoveandTouchFun_2f" "noBreak"
    $ 1870 "b_touch_pos≔A_Prepos_l[A_sel_v]"
    global b_touch_pos=A_Prepos_l[A_sel_v]
    $ 1871 "tilt_deg≔3"
    global tilt_deg=3
    $ 1872 "tilt_deg_ry≔3"
    global tilt_deg_ry=3
    $ 1873 "tilt_deg_rz≔0"
    global tilt_deg_rz=0
    $ 1874 "If b2_left_par"
    if (b2_left_par):
      $ 1875 "b_touch_pos≔pose_trans(b_touch_pos, p[0,0/1000,0,d2r(tilt_deg),d2r(-tilt_deg_ry),d2r(tilt_deg_rz)])"
      global b_touch_pos= pose_trans (b_touch_pos, p[0,0/1000,0,d2r(tilt_deg),d2r(-tilt_deg_ry),d2r(tilt_deg_rz)])
    else:
      $ 1876 "Else" "noBreak"
      $ 1877 "b_touch_pos≔pose_trans(b_touch_pos, p[0,0/1000,0,d2r(tilt_deg),d2r(-tilt_deg_ry),d2r(-tilt_deg_rz)])"
      global b_touch_pos= pose_trans (b_touch_pos, p[0,0/1000,0,d2r(tilt_deg),d2r(-tilt_deg_ry),d2r(-tilt_deg_rz)])
    end
    $ 1878 "MoveL"
    $ 1879 "b_touch_pos" "breakAfter"
    movel(pose_trans(Base, b_touch_pos), a=0.35, v=0.35)
    $ 1880 "Touch_2f"
    $ 1881 "touch_result≔touch_fun_2f(b_touch_pos,b_touch_pos,b2_left_par,b9_touch_sens)"
    global touch_result=touch_fun_2f(b_touch_pos,b_touch_pos,b2_left_par,b9_touch_sens)
    $ 1883 "If b2_left_par"
    if (b2_left_par):
      $ 1884 "touch_result≔pose_trans(touch_result,p[-(Touch_dis)/1000,0,0,0,0,0])"
      global touch_result= pose_trans (touch_result,p[-(Touch_dis)/1000,0,0,0,0,0])
    else:
      $ 1885 "Else" "noBreak"
      $ 1886 "touch_result≔pose_trans(touch_result,p[(Touch_dis)/1000,0,0,0,0,0])"
      global touch_result= pose_trans (touch_result,p[(Touch_dis)/1000,0,0,0,0,0])
    end
    $ 1887 "A_Touch_p[A_sel_v]=touch_result"
    A_Touch_p[A_sel_v]=touch_result
    $ 1888 "If EXT_flag1[3]≟ True "
    if (EXT_flag1[3] ==   True  ):
      $ 1889 "MoveL"
      $ 1890 "manual_tp≔tilt_2f_fun(touch_result,basic_tilt_2f,wv_direction)"
      global manual_tp=tilt_2f_fun(touch_result,basic_tilt_2f,wv_direction)
      $ 1891 "manual_tp≔pose_trans(manual_tp, p[0,0,-10/1000,0,0,0])"
      global manual_tp= pose_trans (manual_tp, p[0,0,-10/1000,0,0,0])
      $ 1892 "manual_tp" "breakAfter"
      movel(pose_trans(Base, manual_tp), a=0.3, v=0.15)
      $ 1893 "Wait: 1.5"
      sleep(1.5)
    end
  end
  def MoveandTouchFun_3f():
    $ 1894 "MoveandTouchFun_3f" "noBreak"
    $ 1895 "b_touch_pos≔A_Prepos_l[A_sel_v]"
    global b_touch_pos=A_Prepos_l[A_sel_v]
    $ 1896 "tilt_deg_ry≔0"
    global tilt_deg_ry=0
    $ 1897 "tilt_deg_rz≔0"
    global tilt_deg_rz=0
    $ 1898 "If b2_left_par"
    if (b2_left_par):
      $ 1899 "tilt_deg≔6"
      global tilt_deg=6
      $ 1900 "b_touch_pos≔pose_trans(b_touch_pos, p[0,0/1000,0,d2r(tilt_deg),d2r(tilt_deg_ry),d2r(tilt_deg_rz)])"
      global b_touch_pos= pose_trans (b_touch_pos, p[0,0/1000,0,d2r(tilt_deg),d2r(tilt_deg_ry),d2r(tilt_deg_rz)])
    else:
      $ 1901 "Else" "noBreak"
      $ 1902 "tilt_deg≔0.5"
      global tilt_deg=0.5
      $ 1903 "b_touch_pos≔pose_trans(b_touch_pos, p[0,0/1000,0,d2r(-tilt_deg),d2r(tilt_deg_ry),d2r(tilt_deg_rz)])"
      global b_touch_pos= pose_trans (b_touch_pos, p[0,0/1000,0,d2r(-tilt_deg),d2r(tilt_deg_ry),d2r(tilt_deg_rz)])
    end
    $ 1914 "move_pre"
    $ 1915 "If (b2_left_par≟ True  and point_dist(A_Prepos_l[A_HOR], A_Prepos_l[A_VL1])>0.032) or (b2_left_par≟ False  and point_dist(A_Prepos_l[A_HOR_R],A_Prepos_l[A_VR1])>0.032)"
    if ((b2_left_par ==   True    and  point_dist(A_Prepos_l[A_HOR], A_Prepos_l[A_VL1])>0.032)  or  (b2_left_par ==   False    and  point_dist(A_Prepos_l[A_HOR_R],A_Prepos_l[A_VR1])>0.032)):
      $ 1916 "if move from home"
      $ 1917 "j_cp≔get_actual_joint_positions()"
      global j_cp= get_actual_joint_positions ()
      $ 1918 "If b2_left_par"
      if (b2_left_par):
        $ 1919 "If norm(b_touch_pos[1]*1000)>300"
        if (norm(b_touch_pos[1]*1000)>300):
          $ 1920 "inner_p≔p[-15/1000,-35/1000,0,0,0,0]"
          global inner_p=p[-15/1000,-35/1000,0,0,0,0]
        else:
          $ 1921 "Else" "noBreak"
          $ 1922 "inner_p≔p[0,0,0,0,0,0]"
          global inner_p=p[0,0,0,0,0,0]
        end
        $ 1923 "j_tp≔get_inverse_kin(pose_add(b_touch_pos,inner_p),qnear=left_j)"
        global j_tp= get_inverse_kin (pose_add(b_touch_pos,inner_p),qnear=left_j)
      else:
        $ 1924 "Else" "noBreak"
        $ 1925 "If norm(b_touch_pos[1]*1000)>300"
        if (norm(b_touch_pos[1]*1000)>300):
          $ 1926 "inner_p≔p[-15/1000,35/1000,0,0,0,0]"
          global inner_p=p[-15/1000,35/1000,0,0,0,0]
        else:
          $ 1927 "Else" "noBreak"
          $ 1928 "inner_p≔p[0,0,0,0,0,0]"
          global inner_p=p[0,0,0,0,0,0]
        end
        $ 1929 "j_tp≔get_inverse_kin(pose_add(b_touch_pos,inner_p),qnear=right_j)"
        global j_tp= get_inverse_kin ( pose_add (b_touch_pos,inner_p),qnear=right_j)
      end
      $ 1930 "j_cp[0]=j_tp[0]"
      j_cp[0]=j_tp[0]
      $ 1931 "j_cp[1]=j_cp[1]+(j_tp[1]-j_cp[1])/2"
      j_cp[1]=j_cp[1]+(j_tp[1]-j_cp[1])/2
      $ 1932 "j_cp[2]=j_cp[2]+(j_tp[2]-j_cp[2])/2.5"
      j_cp[2]=j_cp[2]+(j_tp[2]-j_cp[2])/2.5
      $ 1933 "j_cp[3]=j_cp[3]+(j_tp[3]-j_cp[3])/2.5"
      j_cp[3]=j_cp[3]+(j_tp[3]-j_cp[3])/2.5
      $ 1934 "j_cp[4]=j_cp[4]+(j_tp[4]-j_cp[4])/3"
      j_cp[4]=j_cp[4]+(j_tp[4]-j_cp[4])/3
      $ 1935 "j_cp[5]=j_cp[5]+(j_tp[5]-j_cp[5])/1"
      j_cp[5]=j_cp[5]+(j_tp[5]-j_cp[5])/1
      $ 1936 "MoveJ"
      $ 1937 "j_cp" "breakAfter"
      movej(j_cp, a=1.3962634015954636, v=1.0471975511965976)
      $ 1938 "j_tp≔[j_cp[0],j_cp[1],j_cp[2],j_cp[3],j_tp[4],j_tp[5]]"
      global j_tp=[j_cp[0],j_cp[1],j_cp[2],j_cp[3],j_tp[4],j_tp[5]]
    end
    $ 1941 "MoveL"
    $ 1942 "b_touch_pos" "breakAfter"
    movel(pose_trans(Base, b_touch_pos), a=0.35, v=0.35)
    $ 1945 "touch_3f_down"
    $ 1947 "touch_result≔touch_fun2(b_touch_pos,b2_left_par,b9_touch_sens,b2_par_cd)"
    global touch_result=touch_fun2(b_touch_pos,b2_left_par,b9_touch_sens,b2_par_cd)
    $ 1948 "If Scallup_check≟ False "
    if (Scallup_check ==   False  ):
      $ 1949 "touch_result≔pose_trans(touch_result,p[-(Touch_dis)/1000,0,0,0,0,0])"
      global touch_result= pose_trans (touch_result,p[-(Touch_dis)/1000,0,0,0,0,0])
    else:
      $ 1950 "Else" "noBreak"
      $ 1951 "Scallup_check≔ False "
      global Scallup_check=  False
    end
    $ 1954 "A_Touch_p[A_sel_v]=touch_result"
    A_Touch_p[A_sel_v]=touch_result
    $ 1955 "If EXT_flag1[3]≟ True "
    if (EXT_flag1[3] ==   True  ):
      $ 1956 "MoveL"
      $ 1957 "manual_tp≔tilt_3f_fun(A_Touch_p[A_sel_v],basic_tilt_3f,0)"
      global manual_tp=tilt_3f_fun(A_Touch_p[A_sel_v],basic_tilt_3f,0)
      $ 1958 "manual_tp≔pose_trans(manual_tp, p[0,0,-10/1000,0,0,0])"
      global manual_tp= pose_trans (manual_tp, p[0,0,-10/1000,0,0,0])
      $ 1959 "manual_tp" "breakAfter"
      movel(pose_trans(Base, manual_tp), a=0.3, v=0.15)
      $ 1960 "Wait: 1.5"
      sleep(1.5)
    end
    $ 1961 "touch_3f_up"
    $ 1962 "If A_Prepos_l[A_sel_v_end]≟p[0,0,0,0,0,0]"
    if (A_Prepos_l[A_sel_v_end] == p[0,0,0,0,0,0]):
      $ 1963 "A_Touch_p[A_sel_v_end]=p[0,0,0,0,0,0]"
      A_Touch_p[A_sel_v_end]=p[0,0,0,0,0,0]
    else:
      $ 1964 "Else" "noBreak"
      $ 1965 "b_touch_pos≔A_Prepos_l[A_sel_v_end]"
      global b_touch_pos=A_Prepos_l[A_sel_v_end]
      $ 1966 "MoveL"
      $ 1967 "b_touch_pos" "breakAfter"
      movel(pose_trans(Base, b_touch_pos), a=0.7, v=0.5)
      $ 1968 "touch_result≔touch_fun2(b_touch_pos,b2_left_par,b9_touch_sens)"
      global touch_result=touch_fun2(b_touch_pos,b2_left_par,b9_touch_sens)
      $ 1969 "A_Touch_p[A_sel_v_end]=touch_result"
      A_Touch_p[A_sel_v_end]=touch_result
      $ 1970 "If EXT_flag1[3]≟ True "
      if (EXT_flag1[3] ==   True  ):
        $ 1971 "MoveL"
        $ 1972 "manual_tp≔A_Touch_p[A_sel_v_end]"
        global manual_tp=A_Touch_p[A_sel_v_end]
        $ 1973 "manual_tp≔tilt_3f_fun(A_Touch_p[A_sel_v_end],basic_tilt_3f,0)"
        global manual_tp=tilt_3f_fun(A_Touch_p[A_sel_v_end],basic_tilt_3f,0)
        $ 1974 "manual_tp≔pose_trans(manual_tp, p[0,0,-10/1000,0,0,0])"
        global manual_tp= pose_trans (manual_tp, p[0,0,-10/1000,0,0,0])
        $ 1975 "manual_tp" "breakAfter"
        movel(pose_trans(Base, manual_tp), a=0.3, v=0.15)
        $ 1976 "Wait: 1.5"
        sleep(1.5)
      end
    end
  end
  def weav_welding_3f():
    $ 1980 "weav_welding_3f" "noBreak"
    $ 1981 "If running_trig≟ True "
    global thread_flag_1981=0
    thread Thread_if_1981():
      $ 1982 "inv_inching(inv_inch_time)"
      inv_inching(inv_inch_time)
      $ 1983 "b_touch_pos≔A_Prepos_l[A_sel_v]"
      global b_touch_pos=A_Prepos_l[A_sel_v]
      $ 1984 "move_pre"
      $ 1985 "If (b2_left_par≟ True  and point_dist(A_Prepos_l[A_HOR], A_Prepos_l[A_VL1])>0.032) or (b2_left_par≟ False  and point_dist(A_Prepos_l[A_HOR_R],A_Prepos_l[A_VR1])>0.032)"
      if ((b2_left_par ==   True    and  point_dist(A_Prepos_l[A_HOR], A_Prepos_l[A_VL1])>0.032)  or  (b2_left_par ==   False    and  point_dist(A_Prepos_l[A_HOR_R],A_Prepos_l[A_VR1])>0.032)):
        $ 1986 "if move from home"
        $ 1987 "j_cp≔get_actual_joint_positions()"
        global j_cp= get_actual_joint_positions ()
        $ 1988 "If b2_left_par"
        if (b2_left_par):
          $ 1989 "If norm(b_touch_pos[1]*1000)>300"
          if (norm(b_touch_pos[1]*1000)>300):
            $ 1990 "inner_p≔p[-15/1000,-35/1000,0,0,0,0]"
            global inner_p=p[-15/1000,-35/1000,0,0,0,0]
          else:
            $ 1991 "Else" "noBreak"
            $ 1992 "inner_p≔p[0,0,0,0,0,0]"
            global inner_p=p[0,0,0,0,0,0]
          end
          $ 1993 "j_tp≔get_inverse_kin(pose_add(b_touch_pos,inner_p),qnear=left_j)"
          global j_tp= get_inverse_kin (pose_add(b_touch_pos,inner_p),qnear=left_j)
        else:
          $ 1994 "Else" "noBreak"
          $ 1995 "If norm(b_touch_pos[1]*1000)>300"
          if (norm(b_touch_pos[1]*1000)>300):
            $ 1996 "inner_p≔p[-15/1000,35/1000,0,0,0,0]"
            global inner_p=p[-15/1000,35/1000,0,0,0,0]
          else:
            $ 1997 "Else" "noBreak"
            $ 1998 "inner_p≔p[0,0,0,0,0,0]"
            global inner_p=p[0,0,0,0,0,0]
          end
          $ 1999 "j_tp≔get_inverse_kin(pose_add(b_touch_pos,inner_p),qnear=right_j)"
          global j_tp= get_inverse_kin ( pose_add (b_touch_pos,inner_p),qnear=right_j)
        end
        $ 2000 "j_cp[0]=j_tp[0]"
        j_cp[0]=j_tp[0]
        $ 2001 "j_cp[1]=j_cp[1]+(j_tp[1]-j_cp[1])/2"
        j_cp[1]=j_cp[1]+(j_tp[1]-j_cp[1])/2
        $ 2002 "j_cp[2]=j_cp[2]+(j_tp[2]-j_cp[2])/2.5"
        j_cp[2]=j_cp[2]+(j_tp[2]-j_cp[2])/2.5
        $ 2003 "j_cp[3]=j_cp[3]+(j_tp[3]-j_cp[3])/2.5"
        j_cp[3]=j_cp[3]+(j_tp[3]-j_cp[3])/2.5
        $ 2004 "j_cp[4]=j_cp[4]+(j_tp[4]-j_cp[4])/3"
        j_cp[4]=j_cp[4]+(j_tp[4]-j_cp[4])/3
        $ 2005 "j_cp[5]=j_cp[5]+(j_tp[5]-j_cp[5])/1"
        j_cp[5]=j_cp[5]+(j_tp[5]-j_cp[5])/1
        $ 2006 "MoveJ"
        $ 2007 "j_cp" "breakAfter"
        movej(j_cp, a=1.3962634015954636, v=1.0471975511965976)
        $ 2008 "j_tp≔[j_cp[0],j_cp[1],j_cp[2],j_cp[3],j_tp[4],j_tp[5]]"
        global j_tp=[j_cp[0],j_cp[1],j_cp[2],j_cp[3],j_tp[4],j_tp[5]]
      end
      $ 2011 "If (b2_left_par≟ True ) and (b1_cell_info_L≟A or b1_cell_info_L≟C or b1_cell_info_L≟c) and (A_sel_v≠A_VL2)"
      if ((b2_left_par ==   True  )  and  (b1_cell_info_L == A  or  b1_cell_info_L == C  or  b1_cell_info_L == c)  and  (A_sel_v != A_VL2)):
        $ 2012 "begin_3f_p≔pose_trans(A_Touch_p[A_sel_v],p[(multi_offset_z*(multi_path-1))/1000,0,0,0,0,0])"
        global begin_3f_p= pose_trans (A_Touch_p[A_sel_v],p[(multi_offset_z*(multi_path-1))/1000,0,0,0,0,0])
      else:
        $ 2013 "ElseIf (b2_left_par≟ False ) and (b1_cell_info_R≟A or b1_cell_info_R≟C or b1_cell_info_R≟c) and (A_sel_v≠A_VR2)"
        if ((b2_left_par ==   False  )  and  (b1_cell_info_R == A  or  b1_cell_info_R == C  or  b1_cell_info_R == c)  and  (A_sel_v != A_VR2)):
          $ 2014 "begin_3f_p≔pose_trans(A_Touch_p[A_sel_v],p[(multi_offset_z*(multi_path-1))/1000,0,0,0,0,0])"
          global begin_3f_p= pose_trans (A_Touch_p[A_sel_v],p[(multi_offset_z*(multi_path-1))/1000,0,0,0,0,0])
        else:
          $ 2015 "Else" "noBreak"
          $ 2016 "begin_3f_p≔A_Touch_p[A_sel_v]"
          global begin_3f_p=A_Touch_p[A_sel_v]
        end
      end
      $ 2017 "If b2_left_par≟ False "
      if (b2_left_par ==   False  ):
        $ 2018 "If (b1_cell_info_R≟c or b1_cell_info_R≟d) and A_sel_v≟A_VR2"
        if ((b1_cell_info_R == c  or  b1_cell_info_R == d)  and  A_sel_v == A_VR2):
          $ 2020 "b7_tilt_degree≔[-72,-20,15]"
          global b7_tilt_degree=[-72,-20,15]
          $ 2021 "begin_3f_p=pose_add(begin_3f_p,p[-6/1000,-1.5/1000,0,0,0,0])"
          begin_3f_p= pose_add (begin_3f_p,p[-6/1000,-1.5/1000,0,0,0,0])
          $ 2022 "a2_speed_cpm≔a2_speed_cpm*1"
          global a2_speed_cpm=a2_speed_cpm*1
          $ 2023 "a3_wv_amplitude≔a3_wv_amplitude*1"
          global a3_wv_amplitude=a3_wv_amplitude*1
          $ 2024 "a4_wv_frequency≔a4_wv_frequency*1"
          global a4_wv_frequency=a4_wv_frequency*1
          $ 2025 "b3_dealy_all≔[0,b4_wv_delay2*1,0,b6_wv_delay4*1]"
          global b3_dealy_all=[0,b4_wv_delay2*1,0,b6_wv_delay4*1]
          $ 2026 "a0_volt_ref≔a0_volt_ref*1"
          global a0_volt_ref=a0_volt_ref*1
          $ 2027 "a1_amp_ref≔a1_amp_ref*1"
          global a1_amp_ref=a1_amp_ref*1
          $ 2028 "volt and current"
          $ 2029 "squash_l≔[a0_volt_ref,a1_amp_ref,squash_enable,squash_voltage,squash_current,squash_amp,squash_speed,squash_cycle,waste_cycle,c0_offset_x,c0_offset_z]"
          global squash_l=[a0_volt_ref,a1_amp_ref,squash_enable,squash_voltage,squash_current,squash_amp,squash_speed,squash_cycle,waste_cycle,c0_offset_x,c0_offset_z]
          $ 2030 "set_current_voltage(a1_amp_ref,a0_volt_ref)"
          set_current_voltage(a1_amp_ref,a0_volt_ref)
        end
      end
      $ 2039 "welding_result = line_weaving_tp(begin_3f_p,A_Touch_p[A_sel_v_end],[a8_wv_distance,Circle_Speed,b1_appro_param,a4_wv_frequency,a3_wv_amplitude,b8_wv_type,wv_direction],b7_tilt_degree,b3_dealy_all,a9_wv_weldingon,c3_wv_arc,c7_wv_gap,a5_f_hole,b8_wv_2f,a7_weld_crater,squash_l)"
      welding_result = line_weaving_tp(begin_3f_p,A_Touch_p[A_sel_v_end],[a8_wv_distance,Circle_Speed,b1_appro_param,a4_wv_frequency,a3_wv_amplitude,b8_wv_type,wv_direction],b7_tilt_degree,b3_dealy_all,a9_wv_weldingon,c3_wv_arc,c7_wv_gap,a5_f_hole,b8_wv_2f,a7_weld_crater,squash_l)
      thread_flag_1981 = 1
    end
    if (running_trig ==   True  ):
      global thread_handler_1981=run Thread_if_1981()
      while (thread_flag_1981 == 0):
        if not(running_trig ==   True  ):
          kill thread_handler_1981
          thread_flag_1981 = 2
        else:
          sync()
        end
      end
    else:
      thread_flag_1981 = 2
    end
    $ 2040 "write_port_register(weld_done_137,1)"
    write_port_register(weld_done_137,1)
    $ 2041 "homeing()"
    homeing()
    $ 2042 "If sludge≟1"
    if (sludge == 1):
      $ 2043 "pause_trig≔ True "
      global pause_trig=  True
    end
  end
  def weav_welding_2f():
    $ 2044 "weav_welding_2f" "noBreak"
    $ 2045 "If running_trig≟ True "
    global thread_flag_2045=0
    thread Thread_if_2045():
      $ 2046 "Calculation"
      $ 2047 "If Auto_W_num[Auto_cur_cell]≟31 or Auto_W_num[Auto_cur_cell]≟32 or Auto_W_num[Auto_cur_cell]≟30"
      if (Auto_W_num[Auto_cur_cell] == 31  or  Auto_W_num[Auto_cur_cell] == 32  or  Auto_W_num[Auto_cur_cell] == 30):
        $ 2048 "cal_single"
        $ 2049 "pos_m_path≔A_Touch_p[A_HOR]"
        global pos_m_path=A_Touch_p[A_HOR]
        $ 2050 "pos_m_path_end≔A_Touch_p[A_HOR_R]"
        global pos_m_path_end=A_Touch_p[A_HOR_R]
        $ 2051 "A_middle_weld≔interpolate_pose(pos_m_path, pos_m_path_end,0.5)"
        global A_middle_weld= interpolate_pose (pos_m_path, pos_m_path_end,0.5)
      else:
        $ 2052 "Else" "noBreak"
        $ 2053 "side_offset≔10*current_path"
        global side_offset=10*current_path
        $ 2054 "side_offset≔0"
        global side_offset=0
        $ 2055 "If current_path≟2 or current_path≟4"
        if (current_path == 2  or  current_path == 4):
          $ 2056 "center_offset≔15"
          global center_offset=15
        else:
          $ 2057 "Else" "noBreak"
          $ 2058 "center_offset≔0"
          global center_offset=0
        end
        $ 2059 "cal_multi"
        $ 2060 "pos_m_path≔A_Touch_p[A_HOR]"
        global pos_m_path=A_Touch_p[A_HOR]
        $ 2061 "pos_m_path≔pose_trans(pos_m_path, p[side_offset/1000,0,0,0,0,0])"
        global pos_m_path= pose_trans (pos_m_path, p[side_offset/1000,0,0,0,0,0])
        $ 2062 "pos_m_path_end≔A_Touch_p[A_HOR_R]"
        global pos_m_path_end=A_Touch_p[A_HOR_R]
        $ 2063 "pos_m_path_end≔pose_trans(pos_m_path_end, p[-side_offset/1000,0,0,0,0,0])"
        global pos_m_path_end= pose_trans (pos_m_path_end, p[-side_offset/1000,0,0,0,0,0])
        $ 2064 "A_middle_weld≔interpolate_pose(pos_m_path, pos_m_path_end,0.5)"
        global A_middle_weld= interpolate_pose (pos_m_path, pos_m_path_end,0.5)
        $ 2065 "A_middle_weld≔pose_trans(A_middle_weld, p[-center_offset/1000,0,0,0,0,0])"
        global A_middle_weld= pose_trans (A_middle_weld, p[-center_offset/1000,0,0,0,0,0])
      end
      $ 2066 "gap_half"
      $ 2067 "gap_amp_bak≔c5_wv_gap_y"
      global gap_amp_bak=c5_wv_gap_y
      $ 2068 "gap_speed_bak≔c6_wv_gap_cpm"
      global gap_speed_bak=c6_wv_gap_cpm
      $ 2069 "gap_freq_bak≔c9_wv_gap_freq"
      global gap_freq_bak=c9_wv_gap_freq
      $ 2070 "c5_wv_gap_y≔(a3_wv_amplitude+c5_wv_gap_y)/2"
      global c5_wv_gap_y=(a3_wv_amplitude+c5_wv_gap_y)/2
      $ 2071 "c6_wv_gap_cpm≔(a2_speed_cpm+c6_wv_gap_cpm)/2"
      global c6_wv_gap_cpm=(a2_speed_cpm+c6_wv_gap_cpm)/2
      $ 2072 "c9_wv_gap_freq≔(a4_wv_frequency+c9_wv_gap_freq)/2"
      global c9_wv_gap_freq=(a4_wv_frequency+c9_wv_gap_freq)/2
      $ 2073 "c7_wv_gap≔[c4_gap_enable,c5_wv_gap_y,c6_wv_gap_cpm,c9_wv_gap_freq]"
      global c7_wv_gap=[c4_gap_enable,c5_wv_gap_y,c6_wv_gap_cpm,c9_wv_gap_freq]
      $ 2074 "Weaving"
      $ 2075 "If EXT_flag1[6]"
      if (EXT_flag1[6]):
        $ 2076 "If Auto_W_num[Auto_cur_cell]%10≟1"
        if (Auto_W_num[Auto_cur_cell]%10 == 1):
          $ 2077 "inv_inching(inv_inch_time)"
          inv_inching(inv_inch_time)
          $ 2078 "wv_direction≔1"
          global wv_direction=1
          $ 2079 "welding_result = line_weaving_tp(pos_m_path,A_middle_weld,[a8_wv_distance,Circle_Speed,b1_appro_param,a4_wv_frequency,a3_wv_amplitude,b8_wv_type,wv_direction],b7_tilt_degree,b3_dealy_all,a9_wv_weldingon,c3_wv_arc,c7_wv_gap,a5_f_hole,b8_wv_2f,a7_weld_crater,squash_l)"
          welding_result = line_weaving_tp(pos_m_path,A_middle_weld,[a8_wv_distance,Circle_Speed,b1_appro_param,a4_wv_frequency,a3_wv_amplitude,b8_wv_type,wv_direction],b7_tilt_degree,b3_dealy_all,a9_wv_weldingon,c3_wv_arc,c7_wv_gap,a5_f_hole,b8_wv_2f,a7_weld_crater,squash_l)
          $ 2080 "Wait: 0.5"
          sleep(0.5)
        end
        $ 2081 "If Auto_W_num[Auto_cur_cell]%10≟2"
        if (Auto_W_num[Auto_cur_cell]%10 == 2):
          $ 2082 "inv_inching(inv_inch_time)"
          inv_inching(inv_inch_time)
          $ 2083 "a7_weld_crater≔[d_start_current,d_start_voltage,d_start_time,d_end_current_2,d_end_voltage_2,d_end_time_2,d_lean_degree]"
          global a7_weld_crater=[d_start_current,d_start_voltage,d_start_time,d_end_current_2,d_end_voltage_2,d_end_time_2,d_lean_degree]
          $ 2084 "gap_half_right"
          $ 2085 "a3_wv_amplitude≔gap_amp_bak"
          global a3_wv_amplitude=gap_amp_bak
          $ 2086 "a2_speed_cpm≔gap_speed_bak"
          global a2_speed_cpm=gap_speed_bak
          $ 2087 "a4_wv_frequency≔gap_freq_bak"
          global a4_wv_frequency=gap_freq_bak
          $ 2088 "c7_wv_gap≔[c4_gap_enable,c5_wv_gap_y,c6_wv_gap_cpm,c9_wv_gap_freq]"
          global c7_wv_gap=[c4_gap_enable,c5_wv_gap_y,c6_wv_gap_cpm,c9_wv_gap_freq]
          $ 2089 "wv_direction≔-1"
          global wv_direction=-1
          $ 2090 "A_middle_weld≔feature_offset(A_middle_weld,p[-20/1000,0,0,0,0,0],A_Touch_p[A_sel_v])"
          global A_middle_weld=feature_offset(A_middle_weld,p[-20/1000,0,0,0,0,0],A_Touch_p[A_sel_v])
          $ 2091 "welding_result = line_weaving_tp(pos_m_path_end,A_middle_weld,[a8_wv_distance,Circle_Speed,b1_appro_param,a4_wv_frequency,a3_wv_amplitude,b8_wv_type,wv_direction],b7_tilt_degree,b3_dealy_all,a9_wv_weldingon,c3_wv_arc,c7_wv_gap,a5_f_hole,b8_wv_2f,a7_weld_crater,squash_l)"
          welding_result = line_weaving_tp(pos_m_path_end,A_middle_weld,[a8_wv_distance,Circle_Speed,b1_appro_param,a4_wv_frequency,a3_wv_amplitude,b8_wv_type,wv_direction],b7_tilt_degree,b3_dealy_all,a9_wv_weldingon,c3_wv_arc,c7_wv_gap,a5_f_hole,b8_wv_2f,a7_weld_crater,squash_l)
        end
      else:
        $ 2093 "Else" "noBreak"
        $ 2094 "If Auto_W_num[Auto_cur_cell]%10≟0"
        if (Auto_W_num[Auto_cur_cell]%10 == 0):
          $ 2095 "inv_inching(inv_inch_time)"
          inv_inching(inv_inch_time)
          $ 2096 "wv_direction≔1"
          global wv_direction=1
          $ 2097 "welding_result = line_weaving_tp(pos_m_path,pos_m_path_end,[a8_wv_distance,Circle_Speed,b1_appro_param,a4_wv_frequency,a3_wv_amplitude,b8_wv_type,wv_direction],b7_tilt_degree,b3_dealy_all,a9_wv_weldingon,c3_wv_arc,c7_wv_gap,a5_f_hole,b8_wv_2f,a7_weld_crater,squash_l)"
          welding_result = line_weaving_tp(pos_m_path,pos_m_path_end,[a8_wv_distance,Circle_Speed,b1_appro_param,a4_wv_frequency,a3_wv_amplitude,b8_wv_type,wv_direction],b7_tilt_degree,b3_dealy_all,a9_wv_weldingon,c3_wv_arc,c7_wv_gap,a5_f_hole,b8_wv_2f,a7_weld_crater,squash_l)
        else:
          $ 2098 "Else" "noBreak"
          $ 2099 "write_port_register(142,142)"
          write_port_register(142,142)
          $ 2100 "Halt"
          halt
        end
      end
      thread_flag_2045 = 1
    end
    if (running_trig ==   True  ):
      global thread_handler_2045=run Thread_if_2045()
      while (thread_flag_2045 == 0):
        if not(running_trig ==   True  ):
          kill thread_handler_2045
          thread_flag_2045 = 2
        else:
          sync()
        end
      end
    else:
      thread_flag_2045 = 2
    end
    $ 2101 "write_port_register(weld_done_137,1)"
    write_port_register(weld_done_137,1)
    $ 2102 "MoveL"
    $ 2103 "Direction: Tool Z-"
    global move_thread_flag_2103=0
    thread move_thread_2103():
      enter_critical
      move_thread_flag_2103 = 1
      local towardsPos=calculate_point_to_move_towards(get_forward_kin(), [0.0,0.0,-1.0], 0.03)
      movel(towardsPos, a=1.2, v=0.25)
      move_thread_flag_2103 = 2
      exit_critical
    end
    move_thread_flag_2103 = 0
    move_thread_han_2103 = run move_thread_2103()
    while (True):
      sleep(1.0E-10)
      if (move_thread_flag_2103 > 1):
        join move_thread_han_2103
        $ 2104 "Until (distance)"
        break
      end
      sync()
    end
    $ 2105 "homeing()"
    homeing()
    $ 2106 "If sludge≟1 or (sludge≟2 and current_path>1)"
    if (sludge == 1  or  (sludge == 2  and  current_path>1)):
      $ 2107 "If  not (Auto_W_num[Auto_cur_cell]%10≟1)"
      if (  not  (Auto_W_num[Auto_cur_cell]%10 == 1)):
        $ 2108 "pause_trig≔ True "
        global pause_trig=  True
      end
    end
  end
  def weav_welding_2f_CD():
    $ 2109 "weav_welding_2f_CD" "noBreak"
    $ 2110 "If running_trig≟ True "
    global thread_flag_2110=0
    thread Thread_if_2110():
      $ 2111 "CD_calculation"
      $ 2112 "If (Auto_W_num[Auto_cur_cell]≥100 and Auto_W_num[Auto_cur_cell]<106)  or (Auto_W_num[Auto_cur_cell]≥150 and Auto_W_num[Auto_cur_cell]<156)"
      if ((Auto_W_num[Auto_cur_cell] >= 100  and  Auto_W_num[Auto_cur_cell]<106)   or  (Auto_W_num[Auto_cur_cell] >= 150  and  Auto_W_num[Auto_cur_cell]<156)):
        $ 2113 "cal single"
        $ 2114 "cal_1"
        $ 2115 "pos_m_path_cd≔A_Touch_p[A_sel_v]"
        global pos_m_path_cd=A_Touch_p[A_sel_v]
        $ 2116 "pos_m_p_end_cd≔A_Touch_p[A_sel_v_end]"
        global pos_m_p_end_cd=A_Touch_p[A_sel_v_end]
        $ 2117 "cal_2"
        $ 2118 "pos_m_path≔A_Touch_p[A_sel_v2]"
        global pos_m_path=A_Touch_p[A_sel_v2]
        $ 2119 "pos_m_path_end≔A_Touch_p[A_sel_v_end2]"
        global pos_m_path_end=A_Touch_p[A_sel_v_end2]
        $ 2120 "A_middle_weld≔interpolate_pose(pos_m_path, pos_m_path_end,0.5)"
        global A_middle_weld= interpolate_pose (pos_m_path, pos_m_path_end,0.5)
      else:
        $ 2121 "Else" "noBreak"
        $ 2122 "cal multi"
        $ 2123 "side_offset≔0"
        global side_offset=0
        $ 2124 "If current_path≟2 or current_path≟4"
        if (current_path == 2  or  current_path == 4):
          $ 2125 "center_offset≔15"
          global center_offset=15
        else:
          $ 2126 "Else" "noBreak"
          $ 2127 "center_offset≔0"
          global center_offset=0
        end
        $ 2128 "cal_1_multi"
        $ 2129 "pos_m_path_cd≔A_Touch_p[A_sel_v]"
        global pos_m_path_cd=A_Touch_p[A_sel_v]
        $ 2130 "pos_m_path_cd≔pose_trans(pos_m_path_cd, p[side_offset/1000,0,0,0,0,0])"
        global pos_m_path_cd= pose_trans (pos_m_path_cd, p[side_offset/1000,0,0,0,0,0])
        $ 2131 "pos_m_p_end_cd≔A_Touch_p[A_sel_v_end]"
        global pos_m_p_end_cd=A_Touch_p[A_sel_v_end]
        $ 2132 "pos_m_p_end_cd≔pose_trans(pos_m_p_end_cd, p[-side_offset/1000,0,0,0,0,0])"
        global pos_m_p_end_cd= pose_trans (pos_m_p_end_cd, p[-side_offset/1000,0,0,0,0,0])
        $ 2133 "cal_2_multi"
        $ 2134 "pos_m_path≔A_Touch_p[A_sel_v2]"
        global pos_m_path=A_Touch_p[A_sel_v2]
        $ 2135 "pos_m_path≔pose_trans(pos_m_path, p[side_offset/1000,0,0,0,0,0])"
        global pos_m_path= pose_trans (pos_m_path, p[side_offset/1000,0,0,0,0,0])
        $ 2136 "pos_m_path_end≔A_Touch_p[A_sel_v_end2]"
        global pos_m_path_end=A_Touch_p[A_sel_v_end2]
        $ 2137 "pos_m_path_end≔pose_trans(pos_m_path_end, p[-side_offset/1000,0,0,0,0,0])"
        global pos_m_path_end= pose_trans (pos_m_path_end, p[-side_offset/1000,0,0,0,0,0])
        $ 2138 "A_middle_weld≔interpolate_pose(pos_m_path, pos_m_path_end,0.5)"
        global A_middle_weld= interpolate_pose (pos_m_path, pos_m_path_end,0.5)
        $ 2139 "A_middle_weld≔pose_trans(A_middle_weld, p[center_offset*wv_direction/1000,0,0,0,0,0])"
        global A_middle_weld= pose_trans (A_middle_weld, p[center_offset*wv_direction/1000,0,0,0,0,0])
      end
      $ 2140 "gap_half"
      $ 2141 "gap_amp_bak≔c5_wv_gap_y"
      global gap_amp_bak=c5_wv_gap_y
      $ 2142 "gap_speed_bak≔c6_wv_gap_cpm"
      global gap_speed_bak=c6_wv_gap_cpm
      $ 2143 "gap_freq_bak≔c9_wv_gap_freq"
      global gap_freq_bak=c9_wv_gap_freq
      $ 2144 "c5_wv_gap_y≔(a3_wv_amplitude+c5_wv_gap_y)/2"
      global c5_wv_gap_y=(a3_wv_amplitude+c5_wv_gap_y)/2
      $ 2145 "c6_wv_gap_cpm≔(a2_speed_cpm+c6_wv_gap_cpm)/2"
      global c6_wv_gap_cpm=(a2_speed_cpm+c6_wv_gap_cpm)/2
      $ 2146 "c9_wv_gap_freq≔(a4_wv_frequency+c9_wv_gap_freq)/2"
      global c9_wv_gap_freq=(a4_wv_frequency+c9_wv_gap_freq)/2
      $ 2147 "c7_wv_gap≔[c4_gap_enable,c5_wv_gap_y,c6_wv_gap_cpm,c9_wv_gap_freq]"
      global c7_wv_gap=[c4_gap_enable,c5_wv_gap_y,c6_wv_gap_cpm,c9_wv_gap_freq]
      $ 2148 "If EXT_flag1[4]≟ True  and (b1_cell_info_L≠c and b1_cell_info_L≠d and b1_cell_info_R≠c and b1_cell_info_R≠d)"
      if (EXT_flag1[4] ==   True    and  (b1_cell_info_L != c  and  b1_cell_info_L != d  and  b1_cell_info_R != c  and  b1_cell_info_R != d)):
        $ 2149 "If EXT_flag1[6]"
        if (EXT_flag1[6]):
          $ 2150 "If Auto_W_num[Auto_cur_cell]%10≟1"
          if (Auto_W_num[Auto_cur_cell]%10 == 1):
            $ 2151 "inv_inching(inv_inch_time)"
            inv_inching(inv_inch_time)
            $ 2152 "welding_result = line_weaving_tp_l(pos_m_path_cd,[pos_m_p_end_cd,pos_m_path,A_middle_weld],[a8_wv_distance,Circle_Speed,b1_appro_param,a4_wv_frequency,a3_wv_amplitude,b8_wv_type,wv_direction],b7_tilt_degree,b3_dealy_all,a9_wv_weldingon,c3_wv_arc,c7_wv_gap,a5_f_hole,b8_wv_2f,a7_weld_crater,squash_l)"
            welding_result = line_weaving_tp_l(pos_m_path_cd,[pos_m_p_end_cd,pos_m_path,A_middle_weld],[a8_wv_distance,Circle_Speed,b1_appro_param,a4_wv_frequency,a3_wv_amplitude,b8_wv_type,wv_direction],b7_tilt_degree,b3_dealy_all,a9_wv_weldingon,c3_wv_arc,c7_wv_gap,a5_f_hole,b8_wv_2f,a7_weld_crater,squash_l)
          end
          $ 2153 "If Auto_W_num[Auto_cur_cell]%10≟4"
          if (Auto_W_num[Auto_cur_cell]%10 == 4):
            $ 2154 "inv_inching(inv_inch_time)"
            inv_inching(inv_inch_time)
            $ 2155 "a7_weld_crater≔[d_start_current,d_start_voltage,d_start_time,d_end_current_2,d_end_voltage_2,d_end_time_2,d_lean_degree]"
            global a7_weld_crater=[d_start_current,d_start_voltage,d_start_time,d_end_current_2,d_end_voltage_2,d_end_time_2,d_lean_degree]
            $ 2156 "gap_half"
            $ 2157 "a3_wv_amplitude≔gap_amp_bak"
            global a3_wv_amplitude=gap_amp_bak
            $ 2158 "a2_speed_cpm≔gap_speed_bak"
            global a2_speed_cpm=gap_speed_bak
            $ 2159 "a4_wv_frequency≔gap_freq_bak"
            global a4_wv_frequency=gap_freq_bak
            $ 2160 "c7_wv_gap≔[c4_gap_enable,c5_wv_gap_y,c6_wv_gap_cpm,c9_wv_gap_freq]"
            global c7_wv_gap=[c4_gap_enable,c5_wv_gap_y,c6_wv_gap_cpm,c9_wv_gap_freq]
            $ 2161 "wv_direction≔-1*wv_direction"
            global wv_direction=-1*wv_direction
            $ 2162 "A_middle_weld≔feature_offset(A_middle_weld,p[20*wv_direction/1000,0,0,0,0,0],A_Touch_p[A_sel_v2])"
            global A_middle_weld=feature_offset(A_middle_weld,p[20*wv_direction/1000,0,0,0,0,0],A_Touch_p[A_sel_v2])
            $ 2163 "welding_result = line_weaving_tp(pos_m_path_end,A_middle_weld,[a8_wv_distance,Circle_Speed,b1_appro_param,a4_wv_frequency,a3_wv_amplitude,b8_wv_type,wv_direction],b7_tilt_degree,b3_dealy_all,a9_wv_weldingon,c3_wv_arc,c7_wv_gap,a5_f_hole,b8_wv_2f,a7_weld_crater,squash_l)"
            welding_result = line_weaving_tp(pos_m_path_end,A_middle_weld,[a8_wv_distance,Circle_Speed,b1_appro_param,a4_wv_frequency,a3_wv_amplitude,b8_wv_type,wv_direction],b7_tilt_degree,b3_dealy_all,a9_wv_weldingon,c3_wv_arc,c7_wv_gap,a5_f_hole,b8_wv_2f,a7_weld_crater,squash_l)
          end
        else:
          $ 2164 "Else" "noBreak"
          $ 2165 "If Auto_W_num[Auto_cur_cell]%10≟0"
          if (Auto_W_num[Auto_cur_cell]%10 == 0):
            $ 2166 "inv_inching(inv_inch_time)"
            inv_inching(inv_inch_time)
            $ 2167 "welding_result = line_weaving_tp_l(pos_m_path_cd,[pos_m_p_end_cd,pos_m_path,pos_m_path_end],[a8_wv_distance,Circle_Speed,b1_appro_param,a4_wv_frequency,a3_wv_amplitude,b8_wv_type,wv_direction],b7_tilt_degree,b3_dealy_all,a9_wv_weldingon,c3_wv_arc,c7_wv_gap,a5_f_hole,b8_wv_2f,a7_weld_crater,squash_l)"
            welding_result = line_weaving_tp_l(pos_m_path_cd,[pos_m_p_end_cd,pos_m_path,pos_m_path_end],[a8_wv_distance,Circle_Speed,b1_appro_param,a4_wv_frequency,a3_wv_amplitude,b8_wv_type,wv_direction],b7_tilt_degree,b3_dealy_all,a9_wv_weldingon,c3_wv_arc,c7_wv_gap,a5_f_hole,b8_wv_2f,a7_weld_crater,squash_l)
          else:
            $ 2168 "Else" "noBreak"
            $ 2169 "write_port_register(142,142)"
            write_port_register(142,142)
            $ 2170 "Halt"
            halt
          end
        end
      else:
        $ 2171 "Else" "noBreak"
        $ 2172 "If EXT_flag1[6]"
        if (EXT_flag1[6]):
          $ 2173 "If Auto_W_num[Auto_cur_cell]%10≟2"
          if (Auto_W_num[Auto_cur_cell]%10 == 2):
            $ 2174 "inv_inching(inv_inch_time)"
            inv_inching(inv_inch_time)
            $ 2175 "gap_half"
            $ 2176 "gap_amp_bak≔c5_wv_gap_y"
            global gap_amp_bak=c5_wv_gap_y
            $ 2177 "gap_speed_bak≔c6_wv_gap_cpm"
            global gap_speed_bak=c6_wv_gap_cpm
            $ 2178 "gap_freq_bak≔c9_wv_gap_freq"
            global gap_freq_bak=c9_wv_gap_freq
            $ 2179 "c5_wv_gap_y≔(a3_wv_amplitude+c5_wv_gap_y)/2"
            global c5_wv_gap_y=(a3_wv_amplitude+c5_wv_gap_y)/2
            $ 2180 "c6_wv_gap_cpm≔(a2_speed_cpm+c6_wv_gap_cpm)/2"
            global c6_wv_gap_cpm=(a2_speed_cpm+c6_wv_gap_cpm)/2
            $ 2181 "c9_wv_gap_freq≔(a4_wv_frequency+c9_wv_gap_freq)/2"
            global c9_wv_gap_freq=(a4_wv_frequency+c9_wv_gap_freq)/2
            $ 2182 "c7_wv_gap≔[c4_gap_enable,c5_wv_gap_y,c6_wv_gap_cpm,c9_wv_gap_freq]"
            global c7_wv_gap=[c4_gap_enable,c5_wv_gap_y,c6_wv_gap_cpm,c9_wv_gap_freq]
            $ 2183 "welding_result = line_weaving_tp(pos_m_path_cd,pos_m_p_end_cd,[a8_wv_distance,Circle_Speed,b1_appro_param,a4_wv_frequency,a3_wv_amplitude,b8_wv_type,wv_direction],b7_tilt_degree,b3_dealy_all,a9_wv_weldingon,c3_wv_arc,c7_wv_gap,a5_f_hole,b8_wv_2f,a7_weld_crater,squash_l)"
            welding_result = line_weaving_tp(pos_m_path_cd,pos_m_p_end_cd,[a8_wv_distance,Circle_Speed,b1_appro_param,a4_wv_frequency,a3_wv_amplitude,b8_wv_type,wv_direction],b7_tilt_degree,b3_dealy_all,a9_wv_weldingon,c3_wv_arc,c7_wv_gap,a5_f_hole,b8_wv_2f,a7_weld_crater,squash_l)
            $ 2184 "Wait: 0.5"
            sleep(0.5)
          end
          $ 2185 "If Auto_W_num[Auto_cur_cell]%10≟3"
          if (Auto_W_num[Auto_cur_cell]%10 == 3):
            $ 2186 "inv_inching(inv_inch_time)"
            inv_inching(inv_inch_time)
            $ 2187 "welding_result = line_weaving_tp(pos_m_path,A_middle_weld,[a8_wv_distance,Circle_Speed,b1_appro_param,a4_wv_frequency,a3_wv_amplitude,b8_wv_type,wv_direction],b7_tilt_degree,b3_dealy_all,a9_wv_weldingon,c3_wv_arc,c7_wv_gap,a5_f_hole,b8_wv_2f,a7_weld_crater,squash_l)"
            welding_result = line_weaving_tp(pos_m_path,A_middle_weld,[a8_wv_distance,Circle_Speed,b1_appro_param,a4_wv_frequency,a3_wv_amplitude,b8_wv_type,wv_direction],b7_tilt_degree,b3_dealy_all,a9_wv_weldingon,c3_wv_arc,c7_wv_gap,a5_f_hole,b8_wv_2f,a7_weld_crater,squash_l)
            $ 2188 "Wait: 0.5"
            sleep(0.5)
          end
          $ 2189 "If Auto_W_num[Auto_cur_cell]%10≟4"
          if (Auto_W_num[Auto_cur_cell]%10 == 4):
            $ 2190 "inv_inching(inv_inch_time)"
            inv_inching(inv_inch_time)
            $ 2191 "a7_weld_crater≔[d_start_current,d_start_voltage,d_start_time,d_end_current_2,d_end_voltage_2,d_end_time_2,d_lean_degree]"
            global a7_weld_crater=[d_start_current,d_start_voltage,d_start_time,d_end_current_2,d_end_voltage_2,d_end_time_2,d_lean_degree]
            $ 2192 "gap_half"
            $ 2193 "a3_wv_amplitude≔gap_amp_bak"
            global a3_wv_amplitude=gap_amp_bak
            $ 2194 "a2_speed_cpm≔gap_speed_bak"
            global a2_speed_cpm=gap_speed_bak
            $ 2195 "a4_wv_frequency≔gap_freq_bak"
            global a4_wv_frequency=gap_freq_bak
            $ 2196 "c7_wv_gap≔[c4_gap_enable,c5_wv_gap_y,c6_wv_gap_cpm,c9_wv_gap_freq]"
            global c7_wv_gap=[c4_gap_enable,c5_wv_gap_y,c6_wv_gap_cpm,c9_wv_gap_freq]
            $ 2197 "wv_direction≔-1*wv_direction"
            global wv_direction=-1*wv_direction
            $ 2198 "A_middle_weld≔feature_offset(A_middle_weld,p[20*wv_direction/1000,0,0,0,0,0],A_Touch_p[A_sel_v2])"
            global A_middle_weld=feature_offset(A_middle_weld,p[20*wv_direction/1000,0,0,0,0,0],A_Touch_p[A_sel_v2])
            $ 2199 "welding_result = line_weaving_tp(pos_m_path_end,A_middle_weld,[a8_wv_distance,Circle_Speed,b1_appro_param,a4_wv_frequency,a3_wv_amplitude,b8_wv_type,wv_direction],b7_tilt_degree,b3_dealy_all,a9_wv_weldingon,c3_wv_arc,c7_wv_gap,a5_f_hole,b8_wv_2f,a7_weld_crater,squash_l)"
            welding_result = line_weaving_tp(pos_m_path_end,A_middle_weld,[a8_wv_distance,Circle_Speed,b1_appro_param,a4_wv_frequency,a3_wv_amplitude,b8_wv_type,wv_direction],b7_tilt_degree,b3_dealy_all,a9_wv_weldingon,c3_wv_arc,c7_wv_gap,a5_f_hole,b8_wv_2f,a7_weld_crater,squash_l)
          end
        else:
          $ 2200 "Else" "noBreak"
          $ 2201 "If Auto_W_num[Auto_cur_cell]%10≟2"
          if (Auto_W_num[Auto_cur_cell]%10 == 2):
            $ 2202 "inv_inching(inv_inch_time)"
            inv_inching(inv_inch_time)
            $ 2203 "c7_wv_gap≔[0,c5_wv_gap_y,c6_wv_gap_cpm,c9_wv_gap_freq]"
            global c7_wv_gap=[0,c5_wv_gap_y,c6_wv_gap_cpm,c9_wv_gap_freq]
            $ 2204 "welding_result = line_weaving_tp(pos_m_path_cd,pos_m_p_end_cd,[a8_wv_distance,Circle_Speed,b1_appro_param,a4_wv_frequency,a3_wv_amplitude,b8_wv_type,wv_direction],b7_tilt_degree,b3_dealy_all,a9_wv_weldingon,c3_wv_arc,c7_wv_gap,a5_f_hole,b8_wv_2f,a7_weld_crater,squash_l)"
            welding_result = line_weaving_tp(pos_m_path_cd,pos_m_p_end_cd,[a8_wv_distance,Circle_Speed,b1_appro_param,a4_wv_frequency,a3_wv_amplitude,b8_wv_type,wv_direction],b7_tilt_degree,b3_dealy_all,a9_wv_weldingon,c3_wv_arc,c7_wv_gap,a5_f_hole,b8_wv_2f,a7_weld_crater,squash_l)
            $ 2205 "Wait: 0.5"
            sleep(0.5)
          end
          $ 2206 "If Auto_W_num[Auto_cur_cell]%10≟5"
          if (Auto_W_num[Auto_cur_cell]%10 == 5):
            $ 2207 "inv_inching(inv_inch_time)"
            inv_inching(inv_inch_time)
            $ 2208 "c7_wv_gap≔[c4_gap_enable,c5_wv_gap_y,c6_wv_gap_cpm,c9_wv_gap_freq]"
            global c7_wv_gap=[c4_gap_enable,c5_wv_gap_y,c6_wv_gap_cpm,c9_wv_gap_freq]
            $ 2209 "welding_result = line_weaving_tp(pos_m_path,pos_m_path_end,[a8_wv_distance,Circle_Speed,b1_appro_param,a4_wv_frequency,a3_wv_amplitude,b8_wv_type,wv_direction],b7_tilt_degree,b3_dealy_all,a9_wv_weldingon,c3_wv_arc,c7_wv_gap,a5_f_hole,b8_wv_2f,a7_weld_crater,squash_l)"
            welding_result = line_weaving_tp(pos_m_path,pos_m_path_end,[a8_wv_distance,Circle_Speed,b1_appro_param,a4_wv_frequency,a3_wv_amplitude,b8_wv_type,wv_direction],b7_tilt_degree,b3_dealy_all,a9_wv_weldingon,c3_wv_arc,c7_wv_gap,a5_f_hole,b8_wv_2f,a7_weld_crater,squash_l)
            $ 2210 "Wait: 0.5"
            sleep(0.5)
          end
        end
      end
      thread_flag_2110 = 1
    end
    if (running_trig ==   True  ):
      global thread_handler_2110=run Thread_if_2110()
      while (thread_flag_2110 == 0):
        if not(running_trig ==   True  ):
          kill thread_handler_2110
          thread_flag_2110 = 2
        else:
          sync()
        end
      end
    else:
      thread_flag_2110 = 2
    end
    $ 2211 "write_port_register(weld_done_137,1)"
    write_port_register(weld_done_137,1)
    $ 2215 "wv_direction≔1"
    global wv_direction=1
    $ 2216 "MoveL"
    $ 2217 "Direction: Tool Z-"
    global move_thread_flag_2217=0
    thread move_thread_2217():
      enter_critical
      move_thread_flag_2217 = 1
      local towardsPos=calculate_point_to_move_towards(get_forward_kin(), [0.0,0.0,-1.0], 0.03)
      movel(towardsPos, a=1.2, v=0.25)
      move_thread_flag_2217 = 2
      exit_critical
    end
    move_thread_flag_2217 = 0
    move_thread_han_2217 = run move_thread_2217()
    while (True):
      sleep(1.0E-10)
      if (move_thread_flag_2217 > 1):
        join move_thread_han_2217
        $ 2218 "Until (distance)"
        break
      end
      sync()
    end
    $ 2219 "homeing()"
    homeing()
    $ 2220 "If sludge≟1 or (sludge≟2 and current_path>1)"
    if (sludge == 1  or  (sludge == 2  and  current_path>1)):
      $ 2221 "If  not (Auto_W_num[Auto_cur_cell]%10≟1 or Auto_W_num[Auto_cur_cell]%10≟2 or Auto_W_num[Auto_cur_cell]%10≟3)"
      if (  not  (Auto_W_num[Auto_cur_cell]%10 == 1  or  Auto_W_num[Auto_cur_cell]%10 == 2  or  Auto_W_num[Auto_cur_cell]%10 == 3)):
        $ 2222 "pause_trig≔ True "
        global pause_trig=  True
      end
    end
  end
  def reset_weld_param():
    $ 2223 "reset_weld_param" "noBreak"
    $ 2224 "start_num≔225"
    global start_num=225
    $ 2225 "Loop start_num<237"
    while (start_num<237):
      $ 2226 "write_port_register(start_num,0)"
      write_port_register(start_num,0)
      $ 2227 "start_num≔start_num+1"
      global start_num=start_num+1
    end
    $ 2228 "start_num≔240"
    global start_num=240
    $ 2229 "Loop start_num<256"
    while (start_num<256):
      $ 2230 "write_port_register(start_num,0)"
      write_port_register(start_num,0)
      $ 2231 "start_num≔start_num+1"
      global start_num=start_num+1
    end
  end
  def touch_sub():
    $ 2232 "touch_sub" "noBreak"
    $ 2233 "freedrive"
    $ 2234 "save_timer: Start"
    save_timer_is_counting = True
    $ 2235 "Loop save_tool≟ False  and save_timer≤0.5"
    while (get_tool_digital_in(0) ==   False    and  save_timer <= 0.5):
      $ 2236 "If save_tool≟ False "
      if (get_tool_digital_in(0) ==   False  ):
        $ 2237 "save_timer≔0"
        global save_timer=0
      end
      $ 2238 "If freedrive≟ True  and freedrive_trg≟ False "
      if (get_tool_digital_in(1) ==   True    and  freedrive_trg ==   False  ):
        $ 2239 "'Manual - Freedrive'"
        # 'Manual - Freedrive'
        $ 2240 "freedrive_mode()"
        freedrive_mode()
        $ 2241 "freedrive_trg≔ True "
        global freedrive_trg=  True
      else:
        $ 2242 "ElseIf freedrive≟ False  and freedrive_trg≟ True "
        if (get_tool_digital_in(1) ==   False    and  freedrive_trg ==   True  ):
          $ 2243 "end_freedrive_mode()"
          end_freedrive_mode()
          $ 2244 "freedrive_trg≔ False "
          global freedrive_trg=  False
        end
      end
      $ 2245 "If lamp_trig≟ False "
      if (lamp_trig ==   False  ):
        $ 2246 "lamp_trig≔ True "
        global lamp_trig=  True
      end
      $ 2247 "sync()"
      sync()
    end
    $ 2248 "save_timer: Stop"
    save_timer_is_counting = False
    $ 2249 "save_timer: Reset"
    save_timer = 0
    $ 2250 "write_port_register(touch_done_157,1)"
    write_port_register(touch_done_157,1)
    $ 2251 "Wait read_port_register(touch_done_157)≟0"
    while (not( read_port_register (touch_done_157) == 0)):
      sync()
    end
    $ 2252 "Wait save_tool=LO"
    while (get_tool_digital_in(0) == True):
      sync()
    end
  end
  $ 2 "BeforeStart"
  $ 3 "'RobotVersion'"
  # 'RobotVersion'
  $ 4 "write_port_register(160,47)"
  write_port_register(160,47)
  $ 5 "Teaching for Touch"
  $ 6 "g_current_p≔get_actual_tcp_pose()"
  global g_current_p= get_actual_tcp_pose ()
  $ 7 "MoveJ"
  $ 8 "g_current_p" "breakAfter"
  movej(g_current_p, a=1.3962634015954636, v=1.0471975511965976, r=0.05)
  $ 9 "If  False "
  if (  False  ):
    $ 10 "MoveJ"
    $ 11 "'Home'"
    # 'Home'
    $ 12 "first_p" "breakAfter"
    movej([0.6572912931442261, -1.1853707472430628, -1.1612256209002894, -2.29183799425234, 1.5053011178970337, 2.249363422393799], a=1.3962634015954636, v=1.0471975511965976)
    $ 13 "'3F Left Right'"
    # '3F Left Right'
    $ 14 "left" "breakAfter"
    movej([1.0434843552115187, -1.5100991608390455, -1.7306758129700324, -1.1948061631169296, 1.4628666284450171, 1.848321797880608], a=1.3962634015954636, v=1.0471975511965976)
    $ 15 "right" "breakAfter"
    movej([-0.10351455753530914, -1.3302576856500608, -2.115934992292752, -0.862193753976749, 1.3219395896157813, 2.4264792168573246], a=1.3962634015954636, v=1.0471975511965976)
    $ 16 "'2F Left Right'"
    # '2F Left Right'
    $ 17 "up_left" "breakAfter"
    movej([1.1752926889699076, -1.8019900427886952, -1.320977727654376, -1.5255442863405975, 1.3476341406937622, 2.041365262351603], a=1.3962634015954636, v=1.0471975511965976)
    $ 18 "up_right" "breakAfter"
    movej([-0.490858516659304, -1.5854285429454542, -1.6450882962874376, -1.2830655228732084, 1.6157391701919699, 1.9100727821897805], a=1.3962634015954636, v=1.0471975511965976)
    $ 19 "Packing_pos" "breakAfter"
    movej([1.5877798795700073, -0.0173419157611292, -2.4983108679400843, -1.4065726439105433, 1.626846194267273, 3.0169763565063477], a=1.3962634015954636, v=1.0471975511965976)
    $ 20 "pre_position" "breakAfter"
    movej([1.2637099027633667, -0.695505444203512, -2.0481718222247522, -1.9413569609271448, 2.573765277862549, 1.3775802850723267], a=1.3962634015954636, v=1.0471975511965976)
    $ 21 "middle_pos" "breakAfter"
    movej([-1.8762093791333925, -1.0408674059020342, -1.3551139327963426, -1.843592441478755, 1.9056326083560464, 0.7075109167810423], a=1.3962634015954636, v=1.0471975511965976)
    $ 22 "Mounting_pos" "breakAfter"
    movej([0.6231353085164267, -0.6300961531972575, -0.9034285948871803, -1.770059340221131, 1.417516049558281, 1.7792033261567348], a=1.3962634015954636, v=1.0471975511965976)
    $ 23 "pre_mounting" "breakAfter"
    movej([1.2356762886047363, -0.8703244368182581, -0.942230526600973, -2.3905327955829065, 1.3216267824172974, 2.6514604091644287], a=1.3962634015954636, v=1.0471975511965976)
    $ 24 "'firstly touch center and side, side_L is side touch pose'"
    # 'firstly touch center and side, side_L is side touch pose'
    $ 25 "side_p_L" "breakAfter"
    movej([0.7063748268745771, -1.3604975314992132, -1.990433834727808, -1.0668367667667118, 1.6921872781537495, 1.2509236145111355], a=1.3962634015954636, v=1.0471975511965976)
    $ 26 "side_p_R" "breakAfter"
    movej([0.05431400611996651, -1.4896310011493128, -1.8839471975909632, -1.079590145741598, 1.21127450466156, 2.729013204574585], a=1.3962634015954636, v=1.0471975511965976)
    $ 27 "left_prep_p" "breakAfter"
    movej([0.7465318441390991, -0.9293935934649866, -1.54653245607485, -2.120742146168844, 1.6612900495529175, 1.4639835357666016], a=1.3962634015954636, v=1.0471975511965976)
    $ 28 "right_prep_p" "breakAfter"
    movej([0.2742413878440857, -0.8092182318316858, -1.5809415022479456, -2.0764687697040003, 1.7196621894836426, 2.770606517791748], a=1.3962634015954636, v=1.0471975511965976)
    $ 29 "top_right" "breakAfter"
    movej([-0.02242371234582219, -0.9682979219978707, -1.1486403794481532, -1.814672356578109, 1.0564512116488283, 1.9516847799391646], a=1.3962634015954636, v=1.0471975511965976)
    $ 30 "down_right" "breakAfter"
    movej([-0.10387097169690396, -0.8634965401570085, -1.6224404602167288, -1.9527388322769834, 1.2604034373302166, 1.9362943911099855], a=1.3962634015954636, v=1.0471975511965976)
    $ 31 "way_600_3F_VL1" "breakAfter"
    movej([1.4495428629911409, -0.8691188832486789, -1.6280015865128723, -1.109862842185814, 0.958613460846621, 1.8600136596738885], a=1.3962634015954636, v=1.0471975511965976)
    $ 32 "way_3F_42" "breakAfter"
    movej([0.36805654405146704, -0.7862968504575107, -2.173257016154224, -1.4479178800416523, 0.8821879504915225, 2.8855763836420314], a=1.3962634015954636, v=1.0471975511965976)
    $ 33 "Waypoint_3" "breakAfter"
    movej([1.1380372507706311, -0.9407851141189099, -1.233329099346161, -2.2390373632318763, 1.2601061328687342, 1.8320151492624872], a=1.3962634015954636, v=1.0471975511965976)
  end
  $ 34 "waypoint"
  $ 35 "first_p_wp≔first_p"
  global first_p_wp=p[.431245807847, -.007259877891, .087796870964, 2.814824648791, -.024151220978, 1.380109909682]
  $ 36 "home_pos_j≔get_inverse_kin(first_p,qnear=[0.788235068321228, -1.101443115864889, -1.2219904104815882, -2.3243168036090296, 1.506469488143921, 2.3651483058929443])"
  global home_pos_j= get_inverse_kin (p[.431245807847, -.007259877891, .087796870964, 2.814824648791, -.024151220978, 1.380109909682],qnear=[0.788235068321228, -1.101443115864889, -1.2219904104815882, -2.3243168036090296, 1.506469488143921, 2.3651483058929443])
  $ 37 "left_j≔get_inverse_kin(left,qnear=[1.0260889556530308, -1.5106289215345097, -1.741216762689402, -1.178962336228949, 1.4987324920877318, 1.8103628938054515])"
  global left_j= get_inverse_kin (p[.480496318984, .411279115151, .006998291210, -2.211681476386, -.899147924387, -1.383032568605],qnear=[1.0260889556530308, -1.5106289215345097, -1.741216762689402, -1.178962336228949, 1.4987324920877318, 1.8103628938054515])
  $ 38 "right_j≔get_inverse_kin(right,qnear=[-0.04005625546610858, -1.5553040811514833, -1.9086689348599588, -0.877043115030812, 1.298887151057777, 2.511237649551841])"
  global right_j= get_inverse_kin (p[.475000000000, -.421403215678, .026417194146, 1.917761036827, -1.141682393512, 1.523356199292],qnear=[-0.04005625546610858, -1.5553040811514833, -1.9086689348599588, -0.877043115030812, 1.298887151057777, 2.511237649551841])
  $ 39 "Packing_pos_wp≔Packing_pos"
  global Packing_pos_wp=p[.278714911898, .357008020042, .025408199530, -2.146966801259, .195978635494, -.919933898512]
  $ 40 "left_prep_p_v≔left_prep_p"
  global left_prep_p_v=p[.305384281395, .209992212444, .052849493181, -2.261254200610, -.979668861910, -1.115042887278]
  $ 41 "right_prep_p_v≔right_prep_p"
  global right_prep_p_v=p[.313014950044, -.158485291232, .036185360209, 2.427410851571, -1.381422601175, 1.186756198290]
  $ 42 "pre_position_wp≔pre_position"
  global pre_position_wp=p[-.206981089246, .377817475970, .184983176991, -1.570600793609, -.863923490888, -.089005332274]
  $ 43 "pre_mounting_wp≔pre_mounting"
  global pre_mounting_wp=p[.460443249232, .114922015113, .277198878359, -2.240057458299, .067416497001, -1.614091004704]
  $ 44 "mounting_wp≔Mounting_pos"
  global mounting_wp=p[.365658114054, -.003207132620, .718667154922, -1.220752075696, -.066673751622, -2.363385143972]
  $ 45 "Setting"
  $ 46 "inv_inch_time≔0.4"
  global inv_inch_time=0.4
  $ 47 "a7_cell_bottom≔-50.2"
  global a7_cell_bottom=-50.2
  $ 48 "get_center≔470"
  global get_center=470
  $ 49 "work_touch_dis≔50"
  global work_touch_dis=50
  $ 50 "cd_extra_dis≔6"
  global cd_extra_dis=6
  $ 51 "side_pos_x≔-10"
  global side_pos_x=-10
  $ 52 "sec_touch_dis≔35"
  global sec_touch_dis=35
  $ 53 "Touch_dis≔30"
  global Touch_dis=30
  $ 54 "offset_2f_begin≔5"
  global offset_2f_begin=5
  $ 55 "offset_3f_begin≔5"
  global offset_3f_begin=5
  $ 56 "multi_offset_z≔3"
  global multi_offset_z=3
  $ 57 "simulation_mode≔ False "
  global simulation_mode=  False
  $ 58 "tilt_deg_man≔10"
  global tilt_deg_man=10
  $ 59 "Initialization"
  $ 60 "reset_revolution_counter()"
  reset_revolution_counter()
  $ 61 "get_center_bak≔get_center"
  global get_center_bak=get_center
  $ 62 "welding_program≔ False "
  global welding_program=  False
  $ 63 "vr2_p1≔p[0,0,0,0,0,0]"
  global vr2_p1=p[0,0,0,0,0,0]
  $ 64 "running_trig≔ False "
  global running_trig=  False
  $ 65 "pb_comm_count≔0"
  global pb_comm_count=0
  $ 66 "pendant_hb≔read_port_register(161)"
  global pendant_hb= read_port_register (161)
  $ 67 "pause_trig≔ False "
  global pause_trig=  False
  $ 68 "multi_path≔1"
  global multi_path=1
  $ 69 "reset_trig≔ False "
  global reset_trig=  False
  $ 70 "heartbeat≔0"
  global heartbeat=0
  $ 71 "back_2f≔ False "
  global back_2f=  False
  $ 72 "t_time≔0"
  global t_time=0
  $ 73 "cd_offset≔35"
  global cd_offset=35
  $ 74 "write_port_register(144,0)"
  write_port_register(144,0)
  $ 75 "time_cal_trig≔ False "
  global time_cal_trig=  False
  $ 76 "current_2f≔0"
  global current_2f=0
  $ 77 "A_cur_2f≔0"
  global A_cur_2f=0
  $ 78 "CD_MLR≔ True "
  global CD_MLR=  True
  $ 79 "auto_on≔ False "
  global auto_on=  False
  $ 80 "event_cal_on≔ False "
  global event_cal_on=  False
  $ 81 "event_side_on≔ False "
  global event_side_on=  False
  $ 82 "Auto_trig≔ False "
  global Auto_trig=  False
  $ 83 "lamp_trig≔ False "
  global lamp_trig=  False
  $ 84 "calcu_trig≔ False "
  global calcu_trig=  False
  $ 85 "current_path≔1"
  global current_path=1
  $ 86 "freedrive_trg≔ False "
  global freedrive_trg=  False
  $ 87 "Inch_trg≔ False "
  global Inch_trg=  False
  $ 88 "wv_direction≔1"
  global wv_direction=1
  $ 89 "Move_trig≔ False "
  global Move_trig=  False
  $ 90 "CELL_ROBOT_DIST≔500"
  global CELL_ROBOT_DIST=500
  $ 91 "CELL_WIDTH≔700"
  global CELL_WIDTH=700
  $ 92 "CELL_BOTTOM≔a7_cell_bottom"
  global CELL_BOTTOM=a7_cell_bottom
  $ 93 "scallop_info≔ False "
  global scallop_info=  False
  $ 94 "Carl_info≔ False "
  global Carl_info=  False
  $ 95 "touch_done_2f≔ False "
  global touch_done_2f=  False
  $ 96 "get_pose_side≔0"
  global get_pose_side=0
  $ 97 "get_pose_side_t≔0"
  global get_pose_side_t=0
  $ 98 "ba_trig≔ False "
  global ba_trig=  False
  $ 99 "touch_m_check≔0"
  global touch_m_check=0
  $ 100 "basic_tilt_2f≔[30,5,0]"
  global basic_tilt_2f=[30,5,0]
  $ 102 "basic_tilt_3f≔[0,-27,0]"
  global basic_tilt_3f=[0,-27,0]
  $ 104 "modbus_name"
  $ 105 "weld_done_137≔137"
  global weld_done_137=137
  $ 106 "robot_ready_141≔141"
  global robot_ready_141=141
  $ 107 "cell_3f_2f_151≔151"
  global cell_3f_2f_151=151
  $ 108 "cell_info_152≔152"
  global cell_info_152=152
  $ 109 "weld_req_153≔153"
  global weld_req_153=153
  $ 110 "touch_cell_155≔155"
  global touch_cell_155=155
  $ 111 "touch_num_156≔156"
  global touch_num_156=156
  $ 112 "touch_done_157≔157"
  global touch_done_157=157
  $ 113 "robot_move_163≔163"
  global robot_move_163=163
  $ 114 "robot_pose_164≔164"
  global robot_pose_164=164
  $ 115 "work_type_165≔165"
  global work_type_165=165
  $ 116 "arc_onoff_168≔168"
  global arc_onoff_168=168
  $ 117 "beforeafter_170≔170"
  global beforeafter_170=170
  $ 118 "return_done_240≔240"
  global return_done_240=240
  $ 119 "a0_Job_Mode≔0"
  global a0_Job_Mode=0
  $ 120 "position_3F≔1"
  global position_3F=1
  $ 121 "position_2F≔2"
  global position_2F=2
  $ 122 "cell_par"
  $ 123 "A≔1"
  global A=1
  $ 124 "B≔2"
  global B=2
  $ 125 "C≔3"
  global C=3
  $ 126 "c≔4"
  global c=4
  $ 127 "D≔5"
  global D=5
  $ 128 "d≔6"
  global d=6
  $ 129 "E≔7"
  global E=7
  $ 130 "A_VL1≔1"
  global A_VL1=1
  $ 131 "A_VL2≔2"
  global A_VL2=2
  $ 132 "A_VR1≔3"
  global A_VR1=3
  $ 133 "A_VR2≔4"
  global A_VR2=4
  $ 134 "A_HOR≔5"
  global A_HOR=5
  $ 135 "A_HOR_R≔7"
  global A_HOR_R=7
  $ 136 "A_HOR_ML≔6"
  global A_HOR_ML=6
  $ 137 "A_HOR_MR≔8"
  global A_HOR_MR=8
  $ 138 "A_HOR_M≔9"
  global A_HOR_M=9
  $ 139 "A_VL1_END≔10"
  global A_VL1_END=10
  $ 140 "A_VL2_END≔11"
  global A_VL2_END=11
  $ 141 "A_VR1_END≔12"
  global A_VR1_END=12
  $ 142 "A_VR2_END≔13"
  global A_VR2_END=13
  $ 143 "A_HOR_2path≔14"
  global A_HOR_2path=14
  $ 144 "A_HOR_3path≔15"
  global A_HOR_3path=15
  $ 145 "A_HOR_4path≔16"
  global A_HOR_4path=16
  $ 146 "A_HOR_2path_CD≔17"
  global A_HOR_2path_CD=17
  $ 147 "A_HOR_3path_CD≔18"
  global A_HOR_3path_CD=18
  $ 148 "A_HOR_4path_CD≔19"
  global A_HOR_4path_CD=19
  $ 149 "Script: UR_samho_weaving_V6.7_CB.script"
  wv_wp1 = p[0,0,0,0,0,0]
  dumy_p = p[0,0,0,0,0,0]
  global background_cal = 0
  global background_pose = [dumy_p,dumy_p,dumy_p]
  global background_ready = 0
  global timer_counter = 0
  global timer_counting = False
  global wcr_counter = 0
  global wcr_counting = False
  global get_wcr = False
  global arc_sens_onoff = 0
  global welding_off_t = 55
  global weld_onoff = False
  global isHicomm = True
  global isTouchWCR = True
  global welding_program = False
  global arc_sens_2F = False

  thread thread_timer():
    error_time = 5
    start_gas_time = 2
    while (True):
      if (timer_counting):
        timer_counter = timer_counter + get_steptime()
        write_output_float_register(0,timer_counter)

        get_wcr = read_welder(5)
        weld_onoff = read_welder_control(0)

        welding_off_t = read_port_register(168)
        if(get_wcr):
          global arc_sens_onoff = 1
        else:
          global arc_sens_onoff = 0
        end
        if(get_wcr and welding_off_t == 2 and weld_onoff == True):
          wcr_counter=0
        elif(wcr_counter>(error_time+start_gas_time) and welding_off_t == 2 and weld_onoff == True):
          write_port_register(202,0)
          write_port_register(149,0)
          write_welder(0,False)
          set_standard_digital_out(0,False)
          write_port_register(142,131)
          sleep(0.5)
          halt
        elif(get_wcr == False and welding_off_t == 2 and weld_onoff == True):
          wcr_counter = wcr_counter + get_steptime()
        end
      end
      sync()
    end
  end

  def RTDE_init():
    # timer
    write_output_float_register(0,0)
    # WCR IN
    write_output_float_register(1,0)
    # Welding Current
    write_output_float_register(2,0)
    # Welding Voltage
    write_output_float_register(3,0)
    # X offset
    write_output_float_register(4,0)
    # Z offset
    write_output_float_register(5,0)
    # PLUS Integral
    write_output_float_register(6,0)
    # MINUS Integral
    write_output_float_register(7,0)
    # Standard_Arc_Current
    write_output_float_register(8,0)
    # ALL Integral
    write_output_float_register(9,0)
    # x up
    write_output_float_register(10,0)
    # x ui
    write_output_float_register(11,0)
    # z up
    write_output_float_register(12,0)
    # z ui
    write_output_float_register(13,0)
    # x
    write_output_float_register(14,0)
    # y
    write_output_float_register(15,0)
    # z
    write_output_float_register(16,0)
    # welding on/off polyscope
    write_output_float_register(17,0)
    # touch on/off polyscope
    write_output_float_register(18,0)
    # ratio_t
    write_output_float_register(19,0)
    # get_wcr polyscope
    write_output_float_register(20,0)
    # get_touch polyscope
    write_output_float_register(21,0)
    # write_welder
    write_output_float_register(22,0)
    # MIDDLE_Integral_org
    write_output_float_register(23,0)
    # PLUS Integral_org
    write_output_float_register(24,0)
    # MINUS Integral_org
    write_output_float_register(25,0)

    #init
    global cycle_number = 0
    global cycle_done = False
    global cycle1_plus = 0
    global cycle1_minus = 0
    global cycle1_middle = 0
    global current_to_welding_m = read_port_register(133)
    global voltage_to_welding_m = read_port_register(134)/10
    global c_maxcut = current_to_welding_m*1.2
    global c_mincut = current_to_welding_m*0.8
    global v_maxcut = voltage_to_welding_m*1.2
    global v_mincut = voltage_to_welding_m*0.8
    global Standard_Arc_Current = current_to_welding_m
    global Standard_Arc_voltage = voltage_to_welding_m
    global FB_CURRENT_UR = 0
    global FB_VOLTAGE_UR = 0
    global FB_CURRENT_UR_org = 0
    global FB_VOLTAGE_UR_org = 0
    global one_cycle_p_count = 0
    global one_cycle_m_count = 0
    global one_cycle_p_accum = 0
    global one_cycle_m_accum = 0
    global one_cycle_p_accum_org = 0
    global one_cycle_m_accum_org = 0
    global cal_off_ang_rx = 0
    global cal_off_ang_ry = 0
    global Up = 0
    global Ui = 0
    global Pi_sum = 0
    global Up_z = 0
    global Ui_z = 0
    global Pi_sum_z = 0
    global peak_value = 0
    global ratio_t = 0
    global welding_off_t = 55
    global program_weld_on = False
    global next_path_c = False
    global move_p = [dumy_p,dumy_p,dumy_p]
    global hicomm = True
    global current_on = False
    timer_counter = 0
    sync()
  end

  # get line distance without caring orientation
  def get_line_dist(get_wp1,get_wp2):
    return sqrt((get_wp2[0]-get_wp1[0])*(get_wp2[0]-get_wp1[0])+(get_wp2[1]-get_wp1[1])*(get_wp2[1]-get_wp1[1])+(get_wp2[2]-get_wp1[2])*(get_wp2[2]-get_wp1[2]))
  end

  def plus_minus(num):
    if(num<0):
      return -1
    else:
      return 1
    end
  end

  def get_feature_plane_xz(p1, p2, p3):

    # Step 1. Get the direction vectors
    d12 = [ p2[0]-p1[0], p2[1]-p1[1], p2[2]-p1[2] ]
    d13 = [ p3[0]-p1[0], p3[1]-p1[1], p3[2]-p1[2] ]

    # Step 2. Get the direction vector of Z axis by cross product of d12 and d13
    dy = cross_product(d13, d12)

    # Step 3. Get the X and Z unit direction vectors by normalizing d12 and dz
    temp = norm(d12)
    ux = [ d12[0]/temp, d12[1]/temp, d12[2]/temp ]
    temp = norm(dy)
    uy = [ dy[0]/temp, dy[1]/temp, dy[2]/temp ]

    # Step 4. Get Y unit direction vector by cross product of uz and ux
    uz = cross_product(ux, uy)

    # Step 5. Get the rotation matrix from the unit direction vectors
    rotmat = [ ux[0], ux[1], ux[2], uy[0], uy[1], uy[2], uz[0], uz[1], uz[2] ]

    # Step 6. Get the rotation vector from the rotation matrix
    rotvec = rotmat2rotvec(rotmat)

    # Step 7. Get the feature plane with the origin at p1 and the frame achieved at step 6
    feature_plane = p[ p1[0], p1[1], p1[2], rotvec[0], rotvec[1], rotvec[2] ]

    return feature_plane
  end

  def get_feature_plane_yz(p1, p2, p3):

    # Step 1. Get the direction vectors
    d12 = [ p2[0]-p1[0], p2[1]-p1[1], p2[2]-p1[2] ]
    d13 = [ p3[0]-p1[0], p3[1]-p1[1], p3[2]-p1[2] ]

    # Step 2. Get the direction vector of Z axis by cross product of d12 and d13
    dx = cross_product(d12, d13)

    # Step 3. Get the X and Z unit direction vectors by normalizing d12 and dz
    temp = norm(d12)
    uy = [ d12[0]/temp, d12[1]/temp, d12[2]/temp ]
    temp = norm(dx)
    ux = [ dx[0]/temp, dx[1]/temp, dx[2]/temp ]

    # Step 4. Get Y unit direction vector by cross product of uz and ux
    uz = cross_product(ux, uy)

    # Step 5. Get the rotation matrix from the unit direction vectors
    rotmat = [ ux[0], ux[1], ux[2], uy[0], uy[1], uy[2], uz[0], uz[1], uz[2] ]

    # Step 6. Get the rotation vector from the rotation matrix
    rotvec = rotmat2rotvec(rotmat)

    # Step 7. Get the feature plane with the origin at p1 and the frame achieved at step 6
    feature_plane = p[ p1[0], p1[1], p1[2], rotvec[0], rotvec[1], rotvec[2] ]

    return feature_plane
  end

  def get_feature_plane_xy(p1, p2, p3):

    # Step 1. Get the direction vectors
    d12 = [ p2[0]-p1[0], p2[1]-p1[1], p2[2]-p1[2] ]
    d13 = [ p3[0]-p1[0], p3[1]-p1[1], p3[2]-p1[2] ]

    # Step 2. Get the direction vector of Z axis by cross product of d12 and d13
    dz = cross_product(d12, d13)

    # Step 3. Get the X and Z unit direction vectors by normalizing d12 and dz
    temp = norm(d12)
    ux = [ d12[0]/temp, d12[1]/temp, d12[2]/temp ]
    temp = norm(dz)
    uz = [ dz[0]/temp, dz[1]/temp, dz[2]/temp ]

    # Step 4. Get Y unit direction vector by cross product of uz and ux
    uy = cross_product(uz, ux)

    # Step 5. Get the rotation matrix from the unit direction vectors
    rotmat = [ ux[0], ux[1], ux[2], uy[0], uy[1], uy[2], uz[0], uz[1], uz[2] ]

    # Step 6. Get the rotation vector from the rotation matrix
    rotvec = rotmat2rotvec(rotmat)

    # Step 7. Get the feature plane with the origin at p1 and the frame achieved at step 6
    feature_plane = p[ p1[0], p1[1], p1[2], rotvec[0], rotvec[1], rotvec[2] ]

    return feature_plane
  end

  #### ur_weaving_rev1 by Henry
  #  x_feature = pose_trans(N_Pose,pose_inv(p[0,0,x,0,0,0])
  def feature_offset(fun_pose,fun_offset,fun_plane=p[0,0,0,0,0,0]):
    fun_p_feature = pose_trans ( pose_inv (fun_plane), fun_pose)
    fun_offrot = rotvec2rpy([fun_p_feature[3],fun_p_feature[4],fun_p_feature[5]])
    fun_offset = p[fun_offset[0],fun_offset[1],fun_offset[2],fun_offrot[0]+fun_offset[3],fun_offrot[1]+fun_offset[4],fun_offrot[2]+fun_offset[5]]
    fun_offset_p = p[fun_offset[0],fun_offset[1],fun_offset[2],0,0,0]
    fun_offrpy_rot = rpy2rotvec([fun_offset[3],fun_offset[4],fun_offset[5]])
    fun_offset_rot = p[0,0,0,fun_offrpy_rot[0],fun_offrpy_rot[1],fun_offrpy_rot[2]]
    fun_cal_p = pose_trans(fun_plane,pose_trans(fun_offset_p,fun_p_feature))
    fun_cal_rot = pose_trans(fun_plane,fun_offset_rot)
    result_cal = p[fun_cal_p[0],fun_cal_p[1],fun_cal_p[2],fun_cal_rot[3],fun_cal_rot[4],fun_cal_rot[5]]
    return result_cal
  end

  ## same as changing feature in Move command
  ## Set offset into Plane and move position by it
  def plane_offset(fun_pose,p_offset,fun_plane=p[0,0,0,0,0,0]):
    fun_p_feature = pose_trans ( pose_inv (fun_plane), fun_pose)
    fun_plane = pose_trans(fun_plane,p[p_offset[0],p_offset[1],p_offset[2],0,0,0])
    fun_p_result = pose_trans(pose_trans(fun_plane,p[0,0,0,p_offset[3],p_offset[4],p_offset[5]]),fun_p_feature)
    return fun_p_result
  end

  #  convert from rotation matrix to rotation vector
  ####
  def rotmat2rotvec(rotmat):

    # array to matrix
    r11 = rotmat[0]
    r21 = rotmat[1]
    r31 = rotmat[2]
    r12 = rotmat[3]
    r22 = rotmat[4]
    r32 = rotmat[5]
    r13 = rotmat[6]
    r23 = rotmat[7]
    r33 = rotmat[8]

    # rotation matrix to rotation vector
    theta = acos((r11+r22+r33-1)/2)
    sth = sin(theta)

    if ( (theta > d2r(179.99)) or (theta < d2r(-179.99)) ):
      theta = d2r(180)
      if (r21 < 0):
        if (r31 < 0):
          ux = sqrt((r11+1)/2)
          uy = -sqrt((r22+1)/2)
          uz = -sqrt((r33+1)/2)
        else:
          ux = sqrt((r11+1)/2)
          uy = -sqrt((r22+1)/2)
          uz = sqrt((r33+1)/2)
        end
      else:
        if (r31 < 0):
          ux = sqrt((r11+1)/2)
          uy = sqrt((r22+1)/2)
          uz = -sqrt((r33+1)/2)
        else:
          ux = sqrt((r11+1)/2)
          uy = sqrt((r22+1)/2)
          uz = sqrt((r33+1)/2)
        end
      end
    else:
      ux = (r32-r23)/(2*sth)
      uy = (r13-r31)/(2*sth)
      uz = (r21-r12)/(2*sth)
    end

    rotvec = [(theta*ux),(theta*uy),(theta*uz)]

    return rotvec
  end

  # cross product of two vectors u and v
  ####
  def cross_product(u, v):

    u1 = u[0]
    u2 = u[1]
    u3 = u[2]
    v1 = v[0]
    v2 = v[1]
    v3 = v[2]

    s = [ (u2*v3-u3*v2), (u3*v1-u1*v3), (u1*v2-u2*v1) ]

